LIN {X 0,Y 369.175,Z 240.992,A -85,B 0,C 180,E1 -12786.554,E2 -12786.554} C_VEL
LIN {X 0,Y 369.058,Z 241.013,A -85,B 0,C 180,E1 -12789.863,E2 -12789.863} C_VEL
LIN {X 0,Y 369.03,Z 241.015,A -85,B 0,C 180,E1 -12793.767,E2 -12793.767} C_VEL
LIN {X 0,Y 368.98,Z 241.021,A -85,B 0,C 180,E1 -12797.737,E2 -12797.737} C_VEL
LIN {X 0,Y 368.917,Z 241.027,A -85,B 0,C 180,E1 -12801.214,E2 -12801.214} C_VEL
LIN {X 0,Y 368.943,Z 241.021,A -85,B 0,C 180,E1 -12804.77,E2 -12804.77} C_VEL
LIN {X 0,Y 368.946,Z 241.015,A -85,B 0,C 180,E1 -12807.198,E2 -12807.198} C_VEL
LIN {X 0,Y 368.909,Z 241.02,A -85,B 0,C 180,E1 -12810.948,E2 -12810.948} C_VEL
LIN {X 0,Y 368.906,Z 241.024,A -85,B 0,C 180,E1 -12814.996,E2 -12814.996} C_VEL
LIN {X 0,Y 368.891,Z 241.027,A -85,B 0,C 180,E1 -12818.637,E2 -12818.637} C_VEL
LIN {X 0,Y 368.924,Z 241.033,A -85,B 0,C 180,E1 -12822.016,E2 -12822.016} C_VEL
LIN {X 0,Y 368.976,Z 241.248,A -85,B 0,C 180,E1 -12824.559,E2 -12824.559} C_VEL
LIN {X 0,Y 371.323,Z 251.732,A -85,B 0,C 180,E1 -12827.564,E2 -12827.564} C_VEL
LIN {X 0,Y 372.681,Z 259.06,A -85,B 0,C 180,E1 -12829.517,E2 -12829.517} C_VEL
LIN {X 0,Y 373.416,Z 261.979,A -85,B 0,C 180,E1 -12829.699,E2 -12829.699} C_VEL
LIN {X 0,Y 377.612,Z 280.099,A -85,B 0,C 180,E1 -12830.394,E2 -12830.394} C_VEL
LIN {X 0,Y 378.936,Z 287.781,A -85,B 0,C 180,E1 -12830.649,E2 -12830.649} C_VEL
LIN {X 0,Y 377.335,Z 366.53,A -85,B 0,C 180,E1 -12832.201,E2 -12832.201} C_VEL
LIN {X 0,Y 376.706,Z 379.905,A -85,B 0,C 180,E1 -12832.675,E2 -12832.675} C_VEL
LIN {X 0,Y 375.846,Z 392.955,A -85,B 0,C 180,E1 -12833.369,E2 -12833.369} C_VEL
LIN {X 0,Y 374.825,Z 404.268,A -85,B 0,C 180,E1 -12834.185,E2 -12834.185} C_VEL
LIN {X 0,Y 373.783,Z 414.895,A -85,B 0,C 180,E1 -12835.171,E2 -12835.171} C_VEL
LIN {X 0,Y 372.647,Z 424.936,A -85,B 0,C 180,E1 -12836.329,E2 -12836.329} C_VEL
LIN {X 0,Y 371.476,Z 434.527,A -85,B 0,C 180,E1 -12837.692,E2 -12837.692} C_VEL
LIN {X 0,Y 370.384,Z 443.005,A -85,B 0,C 180,E1 -12839.181,E2 -12839.181} C_VEL
LIN {X 0,Y 369.428,Z 450.372,A -85,B 0,C 180,E1 -12840.788,E2 -12840.788} C_VEL
LIN {X 0,Y 368.76,Z 455.563,A -85,B 0,C 180,E1 -12842.164,E2 -12842.164} C_VEL
LIN {X 0,Y 368.156,Z 460.932,A -85,B 0,C 180,E1 -12843.956,E2 -12843.956} C_VEL
LIN {X 0,Y 367.748,Z 464.988,A -85,B 0,C 180,E1 -12845.739,E2 -12845.739} C_VEL
LIN {X 0,Y 367.429,Z 467.852,A -85,B 0,C 180,E1 -12847.508,E2 -12847.508} C_VEL
LIN {X 0,Y 367.277,Z 469.892,A -85,B 0,C 180,E1 -12849.637,E2 -12849.637} C_VEL
LIN {X 0,Y 367.175,Z 470.375,A -85,B 0,C 180,E1 -12851.01,E2 -12851.01} C_VEL
LIN {X 0,Y 367.211,Z 469.971,A -85,B 0,C 180,E1 -12853.1,E2 -12853.1} C_VEL
LIN {X 0,Y 367.215,Z 468.91,A -85,B 0,C 180,E1 -12854.458,E2 -12854.458} C_VEL
LIN {X 0,Y 367.27,Z 467.556,A -85,B 0,C 180,E1 -12855.595,E2 -12855.595} C_VEL
LIN {X 0,Y 367.534,Z 464.884,A -85,B 0,C 180,E1 -12857.185,E2 -12857.185} C_VEL
LIN {X 0,Y 367.784,Z 460.721,A -85,B 0,C 180,E1 -12858.983,E2 -12858.983} C_VEL
LIN {X 0,Y 368.198,Z 454.637,A -85,B 0,C 180,E1 -12860.939,E2 -12860.939} C_VEL
LIN {X 0,Y 368.734,Z 448.069,A -85,B 0,C 180,E1 -12862.578,E2 -12862.578} C_VEL
LIN {X 0,Y 369.497,Z 439.608,A -85,B 0,C 180,E1 -12864.269,E2 -12864.269} C_VEL
LIN {X 0,Y 370.198,Z 431.102,A -85,B 0,C 180,E1 -12865.645,E2 -12865.645} C_VEL
LIN {X 0,Y 371.129,Z 420.552,A -85,B 0,C 180,E1 -12867.015,E2 -12867.015} C_VEL
LIN {X 0,Y 372.079,Z 409.847,A -85,B 0,C 180,E1 -12868.126,E2 -12868.126} C_VEL
LIN {X 0,Y 372.918,Z 398.589,A -85,B 0,C 180,E1 -12869.055,E2 -12869.055} C_VEL
LIN {X 0,Y 373.573,Z 386.78,A -85,B 0,C 180,E1 -12869.798,E2 -12869.798} C_VEL
LIN {X 0,Y 374.124,Z 374.049,A -85,B 0,C 180,E1 -12870.37,E2 -12870.37} C_VEL
LIN {X 0,Y 374.497,Z 360.971,A -85,B 0,C 180,E1 -12870.739,E2 -12870.739} C_VEL
LIN {X 0,Y 375.543,Z 284.816,A -85,B 0,C 180,E1 -12872.2,E2 -12872.2} C_VEL
LIN {X 0,Y 373.646,Z 274.125,A -85,B 0,C 180,E1 -12872.502,E2 -12872.502} C_VEL
LIN {X 0,Y 372.161,Z 268.743,A -85,B 0,C 180,E1 -12872.748,E2 -12872.748} C_VEL
LIN {X 0,Y 369.987,Z 263.95,A -85,B 0,C 180,E1 -12873.143,E2 -12873.143} C_VEL
LIN {X 0,Y 366.851,Z 258.406,A -85,B 0,C 180,E1 -12873.861,E2 -12873.861} C_VEL
LIN {X 0,Y 364.875,Z 254.78,A -85,B 0,C 180,E1 -12874.526,E2 -12874.526} C_VEL
LIN {X 0,Y 363.761,Z 251.58,A -85,B 0,C 180,E1 -12875.286,E2 -12875.286} C_VEL
LIN {X 0,Y 362.173,Z 242.319,A -85,B 0,C 180,E1 -12877.807,E2 -12877.807} C_VEL
LIN {X 0,Y 362.108,Z 241.901,A -85,B 0,C 180,E1 -12878.034,E2 -12878.034} C_VEL
LIN {X 0,Y 361.968,Z 241.897,A -85,B 0,C 180,E1 -12881.195,E2 -12881.195} C_VEL
LIN {X 0,Y 361.951,Z 241.896,A -85,B 0,C 180,E1 -12884.62,E2 -12884.62} C_VEL
LIN {X 0,Y 361.929,Z 241.891,A -85,B 0,C 180,E1 -12888.1,E2 -12888.1} C_VEL
LIN {X 0,Y 361.89,Z 241.904,A -85,B 0,C 180,E1 -12891.653,E2 -12891.653} C_VEL
LIN {X 0,Y 361.888,Z 241.886,A -85,B 0,C 180,E1 -12895.293,E2 -12895.293} C_VEL
LIN {X 0,Y 361.901,Z 241.889,A -85,B 0,C 180,E1 -12899.044,E2 -12899.044} C_VEL
LIN {X 0,Y 361.874,Z 241.912,A -85,B 0,C 180,E1 -12901.625,E2 -12901.625} C_VEL
LIN {X 0,Y 361.859,Z 241.901,A -85,B 0,C 180,E1 -12905.354,E2 -12905.354} C_VEL
LIN {X 0,Y 361.9,Z 241.903,A -85,B 0,C 180,E1 -12908.42,E2 -12908.42} C_VEL
LIN {X 0,Y 361.871,Z 241.9,A -85,B 0,C 180,E1 -12911.324,E2 -12911.324} C_VEL
LIN {X 0,Y 361.907,Z 241.9,A -85,B 0,C 180,E1 -12914.354,E2 -12914.354} C_VEL
LIN {X 0,Y 361.862,Z 241.909,A -85,B 0,C 180,E1 -12917.563,E2 -12917.563} C_VEL
LIN {X 0,Y 361.846,Z 241.888,A -85,B 0,C 180,E1 -12920.977,E2 -12920.977} C_VEL
LIN {X 0,Y 361.848,Z 241.91,A -85,B 0,C 180,E1 -12924.66,E2 -12924.66} C_VEL
LIN {X 0,Y 361.835,Z 241.91,A -85,B 0,C 180,E1 -12928.378,E2 -12928.378} C_VEL
LIN {X 0,Y 361.901,Z 241.877,A -85,B 0,C 180,E1 -12932.227,E2 -12932.227} C_VEL
LIN {X 0,Y 361.91,Z 241.89,A -85,B 0,C 180,E1 -12934.715,E2 -12934.715} C_VEL
LIN {X 0,Y 361.902,Z 241.908,A -85,B 0,C 180,E1 -12938.769,E2 -12938.769} C_VEL
LIN {X 0,Y 361.954,Z 241.884,A -85,B 0,C 180,E1 -12942.066,E2 -12942.066} C_VEL
LIN {X 0,Y 361.987,Z 241.868,A -85,B 0,C 180,E1 -12946.106,E2 -12946.106} C_VEL
LIN {X 0,Y 362.027,Z 241.885,A -85,B 0,C 180,E1 -12949.943,E2 -12949.943} C_VEL
LIN {X 0,Y 362.144,Z 241.87,A -85,B 0,C 180,E1 -12952.198,E2 -12952.198} C_VEL
LIN {X 0,Y 362.113,Z 241.867,A -85,B 0,C 180,E1 -12954.436,E2 -12954.436} C_VEL
LIN {X 0,Y 362.276,Z 241.826,A -85,B 0,C 180,E1 -12957.782,E2 -12957.782} C_VEL
LIN {X 0,Y 362.423,Z 241.823,A -85,B 0,C 180,E1 -12960.005,E2 -12960.005} C_VEL
LIN {X 0,Y 362.278,Z 241.855,A -85,B 0,C 180,E1 -12962.228,E2 -12962.228} C_VEL
LIN {X 0,Y 362.136,Z 241.866,A -85,B 0,C 180,E1 -12966.692,E2 -12966.692} C_VEL
LIN {X 0,Y 362.002,Z 241.865,A -85,B 0,C 180,E1 -12970.067,E2 -12970.067} C_VEL
LIN {X 0,Y 362.001,Z 241.886,A -85,B 0,C 180,E1 -12973.903,E2 -12973.903} C_VEL
LIN {X 0,Y 361.972,Z 241.893,A -85,B 0,C 180,E1 -12977.943,E2 -12977.943} C_VEL
LIN {X 0,Y 361.867,Z 241.889,A -85,B 0,C 180,E1 -12981.659,E2 -12981.659} C_VEL
LIN {X 0,Y 361.933,Z 241.9,A -85,B 0,C 180,E1 -12985.294,E2 -12985.294} C_VEL
LIN {X 0,Y 361.915,Z 241.897,A -85,B 0,C 180,E1 -12987.783,E2 -12987.783} C_VEL
LIN {X 0,Y 361.846,Z 241.908,A -85,B 0,C 180,E1 -12991.633,E2 -12991.633} C_VEL
LIN {X 0,Y 361.879,Z 241.905,A -85,B 0,C 180,E1 -12995.347,E2 -12995.347} C_VEL
LIN {X 0,Y 361.839,Z 241.91,A -85,B 0,C 180,E1 -12999.022,E2 -12999.022} C_VEL
LIN {X 0,Y 361.845,Z 241.901,A -85,B 0,C 180,E1 -13002.832,E2 -13002.832} C_VEL
LIN {X 0,Y 361.827,Z 241.886,A -85,B 0,C 180,E1 -13005.95,E2 -13005.95} C_VEL
LIN {X 0,Y 361.824,Z 241.914,A -85,B 0,C 180,E1 -13009.251,E2 -13009.251} C_VEL
LIN {X 0,Y 361.875,Z 241.903,A -85,B 0,C 180,E1 -13012.984,E2 -13012.984} C_VEL
LIN {X 0,Y 361.871,Z 241.908,A -85,B 0,C 180,E1 -13016.633,E2 -13016.633} C_VEL
LIN {X 0,Y 361.872,Z 241.911,A -85,B 0,C 180,E1 -13019.672,E2 -13019.672} C_VEL
LIN {X 0,Y 361.988,Z 242.11,A -85,B 0,C 180,E1 -13022.071,E2 -13022.071} C_VEL
LIN {X 0,Y 364.539,Z 255.351,A -85,B 0,C 180,E1 -13025.556,E2 -13025.556} C_VEL
LIN {X 0,Y 364.852,Z 258.893,A -85,B 0,C 180,E1 -13026.441,E2 -13026.441} C_VEL
LIN {X 0,Y 364.083,Z 268.447,A -85,B 0,C 180,E1 -13028.685,E2 -13028.685} C_VEL
LIN {X 0,Y 364.455,Z 271.791,A -85,B 0,C 180,E1 -13028.848,E2 -13028.848} C_VEL
LIN {X 0,Y 368.737,Z 299.58,A -85,B 0,C 180,E1 -13029.617,E2 -13029.617} C_VEL
LIN {X 0,Y 367.555,Z 376.344,A -85,B 0,C 180,E1 -13031.14,E2 -13031.14} C_VEL
LIN {X 0,Y 366.982,Z 389.637,A -85,B 0,C 180,E1 -13031.616,E2 -13031.616} C_VEL
LIN {X 0,Y 366.233,Z 401.838,A -85,B 0,C 180,E1 -13032.264,E2 -13032.264} C_VEL
LIN {X 0,Y 365.407,Z 413.34,A -85,B 0,C 180,E1 -13033.088,E2 -13033.088} C_VEL
LIN {X 0,Y 364.483,Z 425.147,A -85,B 0,C 180,E1 -13034.196,E2 -13034.196} C_VEL
LIN {X 0,Y 363.624,Z 435.74,A -85,B 0,C 180,E1 -13035.448,E2 -13035.448} C_VEL
LIN {X 0,Y 362.713,Z 445.257,A -85,B 0,C 180,E1 -13036.84,E2 -13036.84} C_VEL
LIN {X 0,Y 361.806,Z 454.405,A -85,B 0,C 180,E1 -13038.516,E2 -13038.516} C_VEL
LIN {X 0,Y 361.197,Z 461.769,A -85,B 0,C 180,E1 -13040.198,E2 -13040.198} C_VEL
LIN {X 0,Y 360.82,Z 466.746,A -85,B 0,C 180,E1 -13041.6,E2 -13041.6} C_VEL
LIN {X 0,Y 360.511,Z 471.567,A -85,B 0,C 180,E1 -13043.283,E2 -13043.283} C_VEL
LIN {X 0,Y 360.362,Z 475.253,A -85,B 0,C 180,E1 -13044.966,E2 -13044.966} C_VEL
LIN {X 0,Y 360.281,Z 477.91,A -85,B 0,C 180,E1 -13046.645,E2 -13046.645} C_VEL
LIN {X 0,Y 360.231,Z 479.16,A -85,B 0,C 180,E1 -13047.764,E2 -13047.764} C_VEL
LIN {X 0,Y 360.256,Z 480.002,A -85,B 0,C 180,E1 -13048.883,E2 -13048.883} C_VEL
LIN {X 0,Y 360.282,Z 480.408,A -85,B 0,C 180,E1 -13050,E2 -13050} C_VEL
LIN {X 0,Y 360.255,Z 480.427,A -85,B 0,C 180,E1 -13051.118,E2 -13051.118} C_VEL
LIN {X 0,Y 360.284,Z 479.31,A -85,B 0,C 180,E1 -13053.355,E2 -13053.355} C_VEL
LIN {X 0,Y 360.386,Z 478.118,A -85,B 0,C 180,E1 -13054.474,E2 -13054.474} C_VEL
LIN {X 0,Y 360.587,Z 474.517,A -85,B 0,C 180,E1 -13056.716,E2 -13056.716} C_VEL
LIN {X 0,Y 360.944,Z 470.633,A -85,B 0,C 180,E1 -13058.397,E2 -13058.397} C_VEL
LIN {X 0,Y 361.539,Z 465.636,A -85,B 0,C 180,E1 -13060.076,E2 -13060.076} C_VEL
LIN {X 0,Y 362.3,Z 459.377,A -85,B 0,C 180,E1 -13061.753,E2 -13061.753} C_VEL
LIN {X 0,Y 363.382,Z 451.556,A -85,B 0,C 180,E1 -13063.42,E2 -13063.42} C_VEL
LIN {X 0,Y 364.611,Z 442.258,A -85,B 0,C 180,E1 -13065.015,E2 -13065.015} C_VEL
LIN {X 0,Y 365.623,Z 433.19,A -85,B 0,C 180,E1 -13066.284,E2 -13066.284} C_VEL
LIN {X 0,Y 366.935,Z 423.186,A -85,B 0,C 180,E1 -13067.414,E2 -13067.414} C_VEL
LIN {X 0,Y 368.099,Z 412.726,A -85,B 0,C 180,E1 -13068.363,E2 -13068.363} C_VEL
LIN {X 0,Y 369.239,Z 400.178,A -85,B 0,C 180,E1 -13069.24,E2 -13069.24} C_VEL
LIN {X 0,Y 370.147,Z 387.693,A -85,B 0,C 180,E1 -13069.876,E2 -13069.876} C_VEL
LIN {X 0,Y 370.777,Z 374.729,A -85,B 0,C 180,E1 -13070.311,E2 -13070.311} C_VEL
LIN {X 0,Y 372.168,Z 299.835,A -85,B 0,C 180,E1 -13071.822,E2 -13071.822} C_VEL
LIN {X 0,Y 368.452,Z 280.07,A -85,B 0,C 180,E1 -13072.527,E2 -13072.527} C_VEL
LIN {X 0,Y 365.852,Z 268.462,A -85,B 0,C 180,E1 -13073.019,E2 -13073.019} C_VEL
LIN {X 0,Y 366.141,Z 265.039,A -85,B 0,C 180,E1 -13073.772,E2 -13073.772} C_VEL
LIN {X 0,Y 366.109,Z 261.48,A -85,B 0,C 180,E1 -13074.679,E2 -13074.679} C_VEL
LIN {X 0,Y 364.008,Z 250.919,A -85,B 0,C 180,E1 -13077.605,E2 -13077.605} C_VEL
LIN {X 0,Y 361.939,Z 242.037,A -85,B 0,C 180,E1 -13080.248,E2 -13080.248} C_VEL
LIN {X 0,Y 361.869,Z 241.911,A -85,B 0,C 180,E1 -13084.279,E2 -13084.279} C_VEL
LIN {X 0,Y 361.873,Z 241.909,A -85,B 0,C 180,E1 -13087.22,E2 -13087.22} C_VEL
LIN {X 0,Y 361.827,Z 241.915,A -85,B 0,C 180,E1 -13090.749,E2 -13090.749} C_VEL
LIN {X 0,Y 361.83,Z 241.913,A -85,B 0,C 180,E1 -13094.367,E2 -13094.367} C_VEL
LIN {X 0,Y 361.848,Z 241.893,A -85,B 0,C 180,E1 -13097.566,E2 -13097.566} C_VEL
LIN {X 0,Y 361.844,Z 241.908,A -85,B 0,C 180,E1 -13100.979,E2 -13100.979} C_VEL
LIN {X 0,Y 361.883,Z 241.904,A -85,B 0,C 180,E1 -13104.654,E2 -13104.654} C_VEL
LIN {X 0,Y 361.846,Z 241.905,A -85,B 0,C 180,E1 -13108.367,E2 -13108.367} C_VEL
LIN {X 0,Y 361.878,Z 241.905,A -85,B 0,C 180,E1 -13110.949,E2 -13110.949} C_VEL
LIN {X 0,Y 361.871,Z 241.909,A -85,B 0,C 180,E1 -13114.701,E2 -13114.701} C_VEL
LIN {X 0,Y 361.87,Z 241.906,A -85,B 0,C 180,E1 -13118.341,E2 -13118.341} C_VEL
LIN {X 0,Y 361.929,Z 241.9,A -85,B 0,C 180,E1 -13122.081,E2 -13122.081} C_VEL
LIN {X 0,Y 361.97,Z 241.889,A -85,B 0,C 180,E1 -13125.375,E2 -13125.375} C_VEL
LIN {X 0,Y 361.976,Z 241.887,A -85,B 0,C 180,E1 -13128.8,E2 -13128.8} C_VEL
LIN {X 0,Y 362.099,Z 241.878,A -85,B 0,C 180,E1 -13132.187,E2 -13132.187} C_VEL
LIN {X 0,Y 362.106,Z 241.874,A -85,B 0,C 180,E1 -13134.426,E2 -13134.426} C_VEL
LIN {X 0,Y 362.272,Z 241.854,A -85,B 0,C 180,E1 -13137.771,E2 -13137.771} C_VEL
LIN {X 0,Y 362.402,Z 241.841,A -85,B 0,C 180,E1 -13139.995,E2 -13139.995} C_VEL
LIN {X 0,Y 362.272,Z 241.853,A -85,B 0,C 180,E1 -13142.219,E2 -13142.219} C_VEL
LIN {X 0,Y 362.136,Z 241.868,A -85,B 0,C 180,E1 -13146.681,E2 -13146.681} C_VEL
LIN {X 0,Y 362.023,Z 241.891,A -85,B 0,C 180,E1 -13150.057,E2 -13150.057} C_VEL
LIN {X 0,Y 361.99,Z 241.893,A -85,B 0,C 180,E1 -13153.893,E2 -13153.893} C_VEL
LIN {X 0,Y 361.919,Z 241.904,A -85,B 0,C 180,E1 -13156.929,E2 -13156.929} C_VEL
LIN {X 0,Y 361.882,Z 241.908,A -85,B 0,C 180,E1 -13160.455,E2 -13160.455} C_VEL
LIN {X 0,Y 361.881,Z 241.906,A -85,B 0,C 180,E1 -13164.108,E2 -13164.108} C_VEL
LIN {X 0,Y 361.925,Z 241.884,A -85,B 0,C 180,E1 -13166.716,E2 -13166.716} C_VEL
LIN {X 0,Y 361.853,Z 241.902,A -85,B 0,C 180,E1 -13170.323,E2 -13170.323} C_VEL
LIN {X 0,Y 361.832,Z 241.909,A -85,B 0,C 180,E1 -13174.275,E2 -13174.275} C_VEL
LIN {X 0,Y 361.851,Z 241.91,A -85,B 0,C 180,E1 -13177.22,E2 -13177.22} C_VEL
LIN {X 0,Y 361.879,Z 241.903,A -85,B 0,C 180,E1 -13180.763,E2 -13180.763} C_VEL
LIN {X 0,Y 361.928,Z 242.099,A -85,B 0,C 180,E1 -13184.071,E2 -13184.071} C_VEL
LIN {X 0,Y 364.016,Z 251.258,A -85,B 0,C 180,E1 -13186.778,E2 -13186.778} C_VEL
LIN {X 0,Y 365.668,Z 259.324,A -85,B 0,C 180,E1 -13188.99,E2 -13188.99} C_VEL
LIN {X 0,Y 367.337,Z 264.457,A -85,B 0,C 180,E1 -13189.28,E2 -13189.28} C_VEL
LIN {X 0,Y 371.361,Z 281.98,A -85,B 0,C 180,E1 -13189.972,E2 -13189.972} C_VEL
LIN {X 0,Y 372.513,Z 288.031,A -85,B 0,C 180,E1 -13190.188,E2 -13190.188} C_VEL
LIN {X 0,Y 370.835,Z 366.571,A -85,B 0,C 180,E1 -13191.764,E2 -13191.764} C_VEL
LIN {X 0,Y 370.177,Z 379.944,A -85,B 0,C 180,E1 -13192.245,E2 -13192.245} C_VEL
LIN {X 0,Y 369.34,Z 391.948,A -85,B 0,C 180,E1 -13192.885,E2 -13192.885} C_VEL
LIN {X 0,Y 368.287,Z 403.751,A -85,B 0,C 180,E1 -13193.731,E2 -13193.731} C_VEL
LIN {X 0,Y 367.13,Z 414.957,A -85,B 0,C 180,E1 -13194.782,E2 -13194.782} C_VEL
LIN {X 0,Y 365.735,Z 426.361,A -85,B 0,C 180,E1 -13196.133,E2 -13196.133} C_VEL
LIN {X 0,Y 364.508,Z 435.985,A -85,B 0,C 180,E1 -13197.572,E2 -13197.572} C_VEL
LIN {X 0,Y 363.319,Z 444.544,A -85,B 0,C 180,E1 -13199.162,E2 -13199.162} C_VEL
LIN {X 0,Y 362.23,Z 452.394,A -85,B 0,C 180,E1 -13200.984,E2 -13200.984} C_VEL
LIN {X 0,Y 361.433,Z 458.505,A -85,B 0,C 180,E1 -13202.809,E2 -13202.809} C_VEL
LIN {X 0,Y 360.909,Z 463.203,A -85,B 0,C 180,E1 -13204.633,E2 -13204.633} C_VEL
LIN {X 0,Y 360.543,Z 466.505,A -85,B 0,C 180,E1 -13206.353,E2 -13206.353} C_VEL
LIN {X 0,Y 360.233,Z 468.962,A -85,B 0,C 180,E1 -13208.242,E2 -13208.242} C_VEL
LIN {X 0,Y 360.189,Z 469.949,A -85,B 0,C 180,E1 -13209.463,E2 -13209.463} C_VEL
LIN {X 0,Y 360.092,Z 470.433,A -85,B 0,C 180,E1 -13210.622,E2 -13210.622} C_VEL
LIN {X 0,Y 360.058,Z 470.477,A -85,B 0,C 180,E1 -13211.801,E2 -13211.801} C_VEL
LIN {X 0,Y 360.101,Z 470.105,A -85,B 0,C 180,E1 -13212.977,E2 -13212.977} C_VEL
LIN {X 0,Y 360.121,Z 469.309,A -85,B 0,C 180,E1 -13214.144,E2 -13214.144} C_VEL
LIN {X 0,Y 360.169,Z 468.041,A -85,B 0,C 180,E1 -13215.305,E2 -13215.305} C_VEL
LIN {X 0,Y 360.43,Z 465.192,A -85,B 0,C 180,E1 -13217.113,E2 -13217.113} C_VEL
LIN {X 0,Y 360.659,Z 461.569,A -85,B 0,C 180,E1 -13218.763,E2 -13218.763} C_VEL
LIN {X 0,Y 360.96,Z 456.663,A -85,B 0,C 180,E1 -13220.474,E2 -13220.474} C_VEL
LIN {X 0,Y 361.609,Z 449.814,A -85,B 0,C 180,E1 -13222.337,E2 -13222.337} C_VEL
LIN {X 0,Y 362.215,Z 442.733,A -85,B 0,C 180,E1 -13223.874,E2 -13223.874} C_VEL
LIN {X 0,Y 362.877,Z 434.836,A -85,B 0,C 180,E1 -13225.278,E2 -13225.278} C_VEL
LIN {X 0,Y 363.787,Z 425.158,A -85,B 0,C 180,E1 -13226.677,E2 -13226.677} C_VEL
LIN {X 0,Y 364.814,Z 414.258,A -85,B 0,C 180,E1 -13227.943,E2 -13227.943} C_VEL
LIN {X 0,Y 365.749,Z 402.902,A -85,B 0,C 180,E1 -13228.986,E2 -13228.986} C_VEL
LIN {X 0,Y 366.505,Z 390.434,A -85,B 0,C 180,E1 -13229.862,E2 -13229.862} C_VEL
LIN {X 0,Y 367.136,Z 377.712,A -85,B 0,C 180,E1 -13230.514,E2 -13230.514} C_VEL
LIN {X 0,Y 367.593,Z 365.51,A -85,B 0,C 180,E1 -13230.924,E2 -13230.924} C_VEL
LIN {X 0,Y 368.867,Z 286.373,A -85,B 0,C 180,E1 -13232.484,E2 -13232.484} C_VEL
LIN {X 0,Y 364.244,Z 259.612,A -85,B 0,C 180,E1 -13233.287,E2 -13233.287} C_VEL
LIN {X 0,Y 364.446,Z 256.919,A -85,B 0,C 180,E1 -13233.87,E2 -13233.87} C_VEL
LIN {X 0,Y 363.964,Z 252.7,A -85,B 0,C 180,E1 -13234.985,E2 -13234.985} C_VEL
LIN {X 0,Y 363.761,Z 251.58,A -85,B 0,C 180,E1 -13235.286,E2 -13235.286} C_VEL
LIN {X 0,Y 362.739,Z 249.786,A -85,B 0,C 180,E1 -13235.816,E2 -13235.816} C_VEL
LIN {X 0,Y 356.039,Z 244.929,A -85,B 0,C 180,E1 -13237.513,E2 -13237.513} C_VEL
LIN {X 0,Y 355.136,Z 243.116,A -85,B 0,C 180,E1 -13238.082,E2 -13238.082} C_VEL
LIN {X 0,Y 355.06,Z 242.774,A -85,B 0,C 180,E1 -13238.288,E2 -13238.288} C_VEL
LIN {X 0,Y 354.927,Z 242.773,A -85,B 0,C 180,E1 -13241.42,E2 -13241.42} C_VEL
LIN {X 0,Y 354.899,Z 242.774,A -85,B 0,C 180,E1 -13244.918,E2 -13244.918} C_VEL
LIN {X 0,Y 354.872,Z 242.765,A -85,B 0,C 180,E1 -13248.473,E2 -13248.473} C_VEL
LIN {X 0,Y 354.858,Z 242.78,A -85,B 0,C 180,E1 -13252.104,E2 -13252.104} C_VEL
LIN {X 0,Y 354.858,Z 242.757,A -85,B 0,C 180,E1 -13255.83,E2 -13255.83} C_VEL
LIN {X 0,Y 354.824,Z 242.78,A -85,B 0,C 180,E1 -13259.681,E2 -13259.681} C_VEL
LIN {X 0,Y 354.801,Z 242.789,A -85,B 0,C 180,E1 -13262.331,E2 -13262.331} C_VEL
LIN {X 0,Y 354.81,Z 242.78,A -85,B 0,C 180,E1 -13265.709,E2 -13265.709} C_VEL
LIN {X 0,Y 354.864,Z 242.782,A -85,B 0,C 180,E1 -13269.327,E2 -13269.327} C_VEL
LIN {X 0,Y 354.81,Z 242.77,A -85,B 0,C 180,E1 -13272.881,E2 -13272.881} C_VEL
LIN {X 0,Y 354.841,Z 242.786,A -85,B 0,C 180,E1 -13276.125,E2 -13276.125} C_VEL
LIN {X 0,Y 354.827,Z 242.777,A -85,B 0,C 180,E1 -13279.194,E2 -13279.194} C_VEL
LIN {X 0,Y 354.785,Z 242.773,A -85,B 0,C 180,E1 -13282.406,E2 -13282.406} C_VEL
LIN {X 0,Y 354.786,Z 242.787,A -85,B 0,C 180,E1 -13284.946,E2 -13284.946} C_VEL
LIN {X 0,Y 354.791,Z 242.787,A -85,B 0,C 180,E1 -13288.405,E2 -13288.405} C_VEL
LIN {X 0,Y 354.832,Z 242.759,A -85,B 0,C 180,E1 -13291.625,E2 -13291.625} C_VEL
LIN {X 0,Y 354.88,Z 242.759,A -85,B 0,C 180,E1 -13294.178,E2 -13294.178} C_VEL
LIN {X 0,Y 354.833,Z 242.782,A -85,B 0,C 180,E1 -13297.9,E2 -13297.9} C_VEL
LIN {X 0,Y 354.909,Z 242.761,A -85,B 0,C 180,E1 -13301.896,E2 -13301.896} C_VEL
LIN {X 0,Y 354.932,Z 242.747,A -85,B 0,C 180,E1 -13305.986,E2 -13305.986} C_VEL
LIN {X 0,Y 354.974,Z 242.765,A -85,B 0,C 180,E1 -13309.741,E2 -13309.741} C_VEL
LIN {X 0,Y 355.106,Z 242.747,A -85,B 0,C 180,E1 -13312.042,E2 -13312.042} C_VEL
LIN {X 0,Y 355.087,Z 242.742,A -85,B 0,C 180,E1 -13314.326,E2 -13314.326} C_VEL
LIN {X 0,Y 355.239,Z 242.702,A -85,B 0,C 180,E1 -13317.738,E2 -13317.738} C_VEL
LIN {X 0,Y 355.371,Z 242.701,A -85,B 0,C 180,E1 -13320.005,E2 -13320.005} C_VEL
LIN {X 0,Y 355.241,Z 242.731,A -85,B 0,C 180,E1 -13322.273,E2 -13322.273} C_VEL
LIN {X 0,Y 355.1,Z 242.742,A -85,B 0,C 180,E1 -13326.825,E2 -13326.825} C_VEL
LIN {X 0,Y 354.958,Z 242.742,A -85,B 0,C 180,E1 -13330.269,E2 -13330.269} C_VEL
LIN {X 0,Y 354.946,Z 242.766,A -85,B 0,C 180,E1 -13334.023,E2 -13334.023} C_VEL
LIN {X 0,Y 354.928,Z 242.77,A -85,B 0,C 180,E1 -13338.113,E2 -13338.113} C_VEL
LIN {X 0,Y 354.821,Z 242.768,A -85,B 0,C 180,E1 -13342.111,E2 -13342.111} C_VEL
LIN {X 0,Y 354.905,Z 242.775,A -85,B 0,C 180,E1 -13345.831,E2 -13345.831} C_VEL
LIN {X 0,Y 354.813,Z 242.769,A -85,B 0,C 180,E1 -13349.687,E2 -13349.687} C_VEL
LIN {X 0,Y 354.824,Z 242.787,A -85,B 0,C 180,E1 -13353.687,E2 -13353.687} C_VEL
LIN {X 0,Y 354.802,Z 242.783,A -85,B 0,C 180,E1 -13356.463,E2 -13356.463} C_VEL
LIN {X 0,Y 354.809,Z 242.791,A -85,B 0,C 180,E1 -13359.422,E2 -13359.422} C_VEL
LIN {X 0,Y 354.797,Z 242.778,A -85,B 0,C 180,E1 -13362.87,E2 -13362.87} C_VEL
LIN {X 0,Y 354.776,Z 242.766,A -85,B 0,C 180,E1 -13366.106,E2 -13366.106} C_VEL
LIN {X 0,Y 354.777,Z 242.791,A -85,B 0,C 180,E1 -13369.178,E2 -13369.178} C_VEL
LIN {X 0,Y 354.812,Z 242.78,A -85,B 0,C 180,E1 -13372.407,E2 -13372.407} C_VEL
LIN {X 0,Y 354.824,Z 242.784,A -85,B 0,C 180,E1 -13374.943,E2 -13374.943} C_VEL
LIN {X 0,Y 354.805,Z 242.786,A -85,B 0,C 180,E1 -13378.407,E2 -13378.407} C_VEL
LIN {X 0,Y 354.927,Z 242.945,A -85,B 0,C 180,E1 -13381.8,E2 -13381.8} C_VEL
LIN {X 0,Y 356.95,Z 253.585,A -85,B 0,C 180,E1 -13384.676,E2 -13384.676} C_VEL
LIN {X 0,Y 357.87,Z 259.691,A -85,B 0,C 180,E1 -13386.261,E2 -13386.261} C_VEL
LIN {X 0,Y 357.185,Z 268.454,A -85,B 0,C 180,E1 -13388.351,E2 -13388.351} C_VEL
LIN {X 0,Y 357.698,Z 272.545,A -85,B 0,C 180,E1 -13388.526,E2 -13388.526} C_VEL
LIN {X 0,Y 361.962,Z 301.104,A -85,B 0,C 180,E1 -13389.329,E2 -13389.329} C_VEL
LIN {X 0,Y 360.728,Z 376.236,A -85,B 0,C 180,E1 -13390.843,E2 -13390.843} C_VEL
LIN {X 0,Y 360.138,Z 389.531,A -85,B 0,C 180,E1 -13391.328,E2 -13391.328} C_VEL
LIN {X 0,Y 359.371,Z 401.734,A -85,B 0,C 180,E1 -13391.987,E2 -13391.987} C_VEL
LIN {X 0,Y 358.438,Z 414.047,A -85,B 0,C 180,E1 -13392.896,E2 -13392.896} C_VEL
LIN {X 0,Y 357.495,Z 425.696,A -85,B 0,C 180,E1 -13394.025,E2 -13394.025} C_VEL
LIN {X 0,Y 356.607,Z 436.178,A -85,B 0,C 180,E1 -13395.302,E2 -13395.302} C_VEL
LIN {X 0,Y 355.748,Z 444.724,A -85,B 0,C 180,E1 -13396.578,E2 -13396.578} C_VEL
LIN {X 0,Y 354.787,Z 453.962,A -85,B 0,C 180,E1 -13398.285,E2 -13398.285} C_VEL
LIN {X 0,Y 354.157,Z 461.388,A -85,B 0,C 180,E1 -13400.001,E2 -13400.001} C_VEL
LIN {X 0,Y 353.756,Z 466.418,A -85,B 0,C 180,E1 -13401.431,E2 -13401.431} C_VEL
LIN {X 0,Y 353.43,Z 471.289,A -85,B 0,C 180,E1 -13403.148,E2 -13403.148} C_VEL
LIN {X 0,Y 353.266,Z 475.021,A -85,B 0,C 180,E1 -13404.864,E2 -13404.864} C_VEL
LIN {X 0,Y 353.205,Z 477.722,A -85,B 0,C 180,E1 -13406.578,E2 -13406.578} C_VEL
LIN {X 0,Y 353.156,Z 479.864,A -85,B 0,C 180,E1 -13408.86,E2 -13408.86} C_VEL
LIN {X 0,Y 353.183,Z 480.299,A -85,B 0,C 180,E1 -13410,E2 -13410} C_VEL
LIN {X 0,Y 353.155,Z 480.338,A -85,B 0,C 180,E1 -13411.141,E2 -13411.141} C_VEL
LIN {X 0,Y 353.21,Z 479.266,A -85,B 0,C 180,E1 -13413.423,E2 -13413.423} C_VEL
LIN {X 0,Y 353.302,Z 478.108,A -85,B 0,C 180,E1 -13414.564,E2 -13414.564} C_VEL
LIN {X 0,Y 353.521,Z 474.549,A -85,B 0,C 180,E1 -13416.851,E2 -13416.851} C_VEL
LIN {X 0,Y 353.921,Z 470.708,A -85,B 0,C 180,E1 -13418.565,E2 -13418.565} C_VEL
LIN {X 0,Y 354.55,Z 465.758,A -85,B 0,C 180,E1 -13420.277,E2 -13420.277} C_VEL
LIN {X 0,Y 355.346,Z 459.552,A -85,B 0,C 180,E1 -13421.986,E2 -13421.986} C_VEL
LIN {X 0,Y 356.487,Z 451.818,A -85,B 0,C 180,E1 -13423.685,E2 -13423.685} C_VEL
LIN {X 0,Y 357.747,Z 442.831,A -85,B 0,C 180,E1 -13425.271,E2 -13425.271} C_VEL
LIN {X 0,Y 358.842,Z 433.631,A -85,B 0,C 180,E1 -13426.601,E2 -13426.601} C_VEL
LIN {X 0,Y 360.202,Z 423.754,A -85,B 0,C 180,E1 -13427.75,E2 -13427.75} C_VEL
LIN {X 0,Y 361.409,Z 413.501,A -85,B 0,C 180,E1 -13428.715,E2 -13428.715} C_VEL
LIN {X 0,Y 362.607,Z 401.273,A -85,B 0,C 180,E1 -13429.606,E2 -13429.606} C_VEL
LIN {X 0,Y 363.576,Z 388.474,A -85,B 0,C 180,E1 -13430.288,E2 -13430.288} C_VEL
LIN {X 0,Y 364.257,Z 376.163,A -85,B 0,C 180,E1 -13430.728,E2 -13430.728} C_VEL
LIN {X 0,Y 365.781,Z 300.95,A -85,B 0,C 180,E1 -13432.278,E2 -13432.278} C_VEL
LIN {X 0,Y 362.169,Z 281.629,A -85,B 0,C 180,E1 -13432.987,E2 -13432.987} C_VEL
LIN {X 0,Y 359.149,Z 268.362,A -85,B 0,C 180,E1 -13433.565,E2 -13433.565} C_VEL
LIN {X 0,Y 359.368,Z 264.123,A -85,B 0,C 180,E1 -13434.556,E2 -13434.556} C_VEL
LIN {X 0,Y 357.652,Z 254.814,A -85,B 0,C 180,E1 -13437.162,E2 -13437.162} C_VEL
LIN {X 0,Y 355.202,Z 244.239,A -85,B 0,C 180,E1 -13440.3,E2 -13440.3} C_VEL
LIN {X 0,Y 354.84,Z 242.816,A -85,B 0,C 180,E1 -13440.83,E2 -13440.83} C_VEL
LIN {X 0,Y 354.822,Z 242.784,A -85,B 0,C 180,E1 -13443.701,E2 -13443.701} C_VEL
LIN {X 0,Y 354.81,Z 242.786,A -85,B 0,C 180,E1 -13446.458,E2 -13446.458} C_VEL
LIN {X 0,Y 354.783,Z 242.784,A -85,B 0,C 180,E1 -13449.411,E2 -13449.411} C_VEL
LIN {X 0,Y 354.799,Z 242.777,A -85,B 0,C 180,E1 -13452.864,E2 -13452.864} C_VEL
LIN {X 0,Y 354.78,Z 242.784,A -85,B 0,C 180,E1 -13456.101,E2 -13456.101} C_VEL
LIN {X 0,Y 354.799,Z 242.789,A -85,B 0,C 180,E1 -13459.176,E2 -13459.176} C_VEL
LIN {X 0,Y 354.813,Z 242.786,A -85,B 0,C 180,E1 -13462.402,E2 -13462.402} C_VEL
LIN {X 0,Y 354.82,Z 242.784,A -85,B 0,C 180,E1 -13464.937,E2 -13464.937} C_VEL
LIN {X 0,Y 354.802,Z 242.782,A -85,B 0,C 180,E1 -13468.403,E2 -13468.403} C_VEL
LIN {X 0,Y 354.808,Z 242.781,A -85,B 0,C 180,E1 -13471.611,E2 -13471.611} C_VEL
LIN {X 0,Y 354.814,Z 242.781,A -85,B 0,C 180,E1 -13475.416,E2 -13475.416} C_VEL
LIN {X 0,Y 354.835,Z 242.782,A -85,B 0,C 180,E1 -13479.109,E2 -13479.109} C_VEL
LIN {X 0,Y 354.889,Z 242.777,A -85,B 0,C 180,E1 -13482.715,E2 -13482.715} C_VEL
LIN {X 0,Y 354.959,Z 242.768,A -85,B 0,C 180,E1 -13486.251,E2 -13486.251} C_VEL
LIN {X 0,Y 354.961,Z 242.762,A -85,B 0,C 180,E1 -13489.731,E2 -13489.731} C_VEL
LIN {X 0,Y 355.11,Z 242.746,A -85,B 0,C 180,E1 -13493.175,E2 -13493.175} C_VEL
LIN {X 0,Y 355.234,Z 242.73,A -85,B 0,C 180,E1 -13497.727,E2 -13497.727} C_VEL
LIN {X 0,Y 355.353,Z 242.719,A -85,B 0,C 180,E1 -13499.995,E2 -13499.995} C_VEL
LIN {X 0,Y 355.234,Z 242.728,A -85,B 0,C 180,E1 -13502.262,E2 -13502.262} C_VEL
LIN {X 0,Y 355.1,Z 242.743,A -85,B 0,C 180,E1 -13506.814,E2 -13506.814} C_VEL
LIN {X 0,Y 354.97,Z 242.768,A -85,B 0,C 180,E1 -13510.259,E2 -13510.259} C_VEL
LIN {X 0,Y 354.935,Z 242.773,A -85,B 0,C 180,E1 -13514.013,E2 -13514.013} C_VEL
LIN {X 0,Y 354.879,Z 242.778,A -85,B 0,C 180,E1 -13518.086,E2 -13518.086} C_VEL
LIN {X 0,Y 354.822,Z 242.781,A -85,B 0,C 180,E1 -13522.1,E2 -13522.1} C_VEL
LIN {X 0,Y 354.883,Z 242.761,A -85,B 0,C 180,E1 -13525.822,E2 -13525.822} C_VEL
LIN {X 0,Y 354.799,Z 242.785,A -85,B 0,C 180,E1 -13529.676,E2 -13529.676} C_VEL
LIN {X 0,Y 354.784,Z 242.79,A -85,B 0,C 180,E1 -13533.696,E2 -13533.696} C_VEL
LIN {X 0,Y 354.78,Z 242.792,A -85,B 0,C 180,E1 -13536.453,E2 -13536.453} C_VEL
LIN {X 0,Y 354.799,Z 242.79,A -85,B 0,C 180,E1 -13539.418,E2 -13539.418} C_VEL
LIN {X 0,Y 354.83,Z 242.783,A -85,B 0,C 180,E1 -13542.874,E2 -13542.874} C_VEL
LIN {X 0,Y 354.903,Z 243.018,A -85,B 0,C 180,E1 -13543.589,E2 -13543.589} C_VEL
LIN {X 0,Y 357.062,Z 252.501,A -85,B 0,C 180,E1 -13546.457,E2 -13546.457} C_VEL
LIN {X 0,Y 358.533,Z 259.431,A -85,B 0,C 180,E1 -13548.402,E2 -13548.402} C_VEL
LIN {X 0,Y 360.839,Z 265.481,A -85,B 0,C 180,E1 -13548.779,E2 -13548.779} C_VEL
LIN {X 0,Y 364.861,Z 282.541,A -85,B 0,C 180,E1 -13549.484,E2 -13549.484} C_VEL
LIN {X 0,Y 366.103,Z 289.065,A -85,B 0,C 180,E1 -13549.724,E2 -13549.724} C_VEL
LIN {X 0,Y 364.373,Z 366.84,A -85,B 0,C 180,E1 -13551.314,E2 -13551.314} C_VEL
LIN {X 0,Y 363.691,Z 380.152,A -85,B 0,C 180,E1 -13551.802,E2 -13551.802} C_VEL
LIN {X 0,Y 362.731,Z 393.202,A -85,B 0,C 180,E1 -13552.519,E2 -13552.519} C_VEL
LIN {X 0,Y 361.488,Z 405.594,A -85,B 0,C 180,E1 -13553.458,E2 -13553.458} C_VEL
LIN {X 0,Y 360.206,Z 417.289,A -85,B 0,C 180,E1 -13554.619,E2 -13554.619} C_VEL
LIN {X 0,Y 358.862,Z 427.57,A -85,B 0,C 180,E1 -13555.903,E2 -13555.903} C_VEL
LIN {X 0,Y 357.664,Z 436.404,A -85,B 0,C 180,E1 -13557.273,E2 -13557.273} C_VEL
LIN {X 0,Y 356.467,Z 444.617,A -85,B 0,C 180,E1 -13558.833,E2 -13558.833} C_VEL
LIN {X 0,Y 355.302,Z 452.643,A -85,B 0,C 180,E1 -13560.735,E2 -13560.735} C_VEL
LIN {X 0,Y 354.592,Z 457.679,A -85,B 0,C 180,E1 -13562.24,E2 -13562.24} C_VEL
LIN {X 0,Y 353.977,Z 462.623,A -85,B 0,C 180,E1 -13564.1,E2 -13564.1} C_VEL
LIN {X 0,Y 353.49,Z 466.538,A -85,B 0,C 180,E1 -13566.124,E2 -13566.124} C_VEL
LIN {X 0,Y 353.207,Z 468.761,A -85,B 0,C 180,E1 -13567.786,E2 -13567.786} C_VEL
LIN {X 0,Y 353.11,Z 470.006,A -85,B 0,C 180,E1 -13569.279,E2 -13569.279} C_VEL
LIN {X 0,Y 352.956,Z 470.621,A -85,B 0,C 180,E1 -13571.422,E2 -13571.422} C_VEL
LIN {X 0,Y 353.01,Z 470.24,A -85,B 0,C 180,E1 -13572.84,E2 -13572.84} C_VEL
LIN {X 0,Y 353.044,Z 468.519,A -85,B 0,C 180,E1 -13575.001,E2 -13575.001} C_VEL
LIN {X 0,Y 353.332,Z 465.494,A -85,B 0,C 180,E1 -13577.035,E2 -13577.035} C_VEL
LIN {X 0,Y 353.613,Z 460.942,A -85,B 0,C 180,E1 -13579.116,E2 -13579.116} C_VEL
LIN {X 0,Y 353.995,Z 455.837,A -85,B 0,C 180,E1 -13580.861,E2 -13580.861} C_VEL
LIN {X 0,Y 354.592,Z 449.515,A -85,B 0,C 180,E1 -13582.57,E2 -13582.57} C_VEL
LIN {X 0,Y 355.323,Z 441.343,A -85,B 0,C 180,E1 -13584.324,E2 -13584.324} C_VEL
LIN {X 0,Y 356.032,Z 433.143,A -85,B 0,C 180,E1 -13585.754,E2 -13585.754} C_VEL
LIN {X 0,Y 357.017,Z 423.105,A -85,B 0,C 180,E1 -13587.179,E2 -13587.179} C_VEL
LIN {X 0,Y 358.054,Z 412.586,A -85,B 0,C 180,E1 -13588.369,E2 -13588.369} C_VEL
LIN {X 0,Y 358.94,Z 401.659,A -85,B 0,C 180,E1 -13589.354,E2 -13589.354} C_VEL
LIN {X 0,Y 359.727,Z 389.395,A -85,B 0,C 180,E1 -13590.21,E2 -13590.21} C_VEL
LIN {X 0,Y 360.28,Z 377.835,A -85,B 0,C 180,E1 -13590.803,E2 -13590.803} C_VEL
LIN {X 0,Y 360.743,Z 364.45,A -85,B 0,C 180,E1 -13591.25,E2 -13591.25} C_VEL
LIN {X 0,Y 362.08,Z 287.214,A -85,B 0,C 180,E1 -13592.799,E2 -13592.799} C_VEL
LIN {X 0,Y 357.38,Z 259.78,A -85,B 0,C 180,E1 -13593.629,E2 -13593.629} C_VEL
LIN {X 0,Y 357.452,Z 258.137,A -85,B 0,C 180,E1 -13593.946,E2 -13593.946} C_VEL
LIN {X 0,Y 356.976,Z 253.888,A -85,B 0,C 180,E1 -13595.082,E2 -13595.082} C_VEL
LIN {X 0,Y 355.395,Z 244.502,A -85,B 0,C 180,E1 -13597.67,E2 -13597.67} C_VEL
LIN {X 0,Y 355.136,Z 243.116,A -85,B 0,C 180,E1 -13598.082,E2 -13598.082} C_VEL
LIN {X 0,Y 354.808,Z 242.788,A -85,B 0,C 180,E1 -13598.52,E2 -13598.52} C_VEL
LIN {X 0,Y 352.554,Z 243.069,A -85,B 0,C 180,E1 -13599.89,E2 -13599.89} C_VEL
LIN {X 0,Y 348.94,Z 243.698,A -85,B 0,C 180,E1 -13601.774,E2 -13601.774} C_VEL
LIN {X 0,Y 347.953,Z 243.662,A -85,B 0,C 180,E1 -13602.761,E2 -13602.761} C_VEL
LIN {X 0,Y 347.877,Z 243.651,A -85,B 0,C 180,E1 -13603.095,E2 -13603.095} C_VEL
LIN {X 0,Y 347.815,Z 243.661,A -85,B 0,C 180,E1 -13606.432,E2 -13606.432} C_VEL
LIN {X 0,Y 347.822,Z 243.639,A -85,B 0,C 180,E1 -13608.862,E2 -13608.862} C_VEL
LIN {X 0,Y 347.808,Z 243.66,A -85,B 0,C 180,E1 -13612.576,E2 -13612.576} C_VEL
LIN {X 0,Y 347.79,Z 243.631,A -85,B 0,C 180,E1 -13616.395,E2 -13616.395} C_VEL
LIN {X 0,Y 347.757,Z 243.662,A -85,B 0,C 180,E1 -13620.347,E2 -13620.347} C_VEL
LIN {X 0,Y 347.746,Z 243.671,A -85,B 0,C 180,E1 -13623.07,E2 -13623.07} C_VEL
LIN {X 0,Y 347.771,Z 243.659,A -85,B 0,C 180,E1 -13626.078,E2 -13626.078} C_VEL
LIN {X 0,Y 347.789,Z 243.66,A -85,B 0,C 180,E1 -13628.787,E2 -13628.787} C_VEL
LIN {X 0,Y 347.788,Z 243.647,A -85,B 0,C 180,E1 -13631.824,E2 -13631.824} C_VEL
LIN {X 0,Y 347.818,Z 243.653,A -85,B 0,C 180,E1 -13635.007,E2 -13635.007} C_VEL
LIN {X 0,Y 347.756,Z 243.66,A -85,B 0,C 180,E1 -13638.395,E2 -13638.395} C_VEL
LIN {X 0,Y 347.751,Z 243.644,A -85,B 0,C 180,E1 -13642.015,E2 -13642.015} C_VEL
LIN {X 0,Y 347.718,Z 243.667,A -85,B 0,C 180,E1 -13645.541,E2 -13645.541} C_VEL
LIN {X 0,Y 347.74,Z 243.667,A -85,B 0,C 180,E1 -13648.308,E2 -13648.308} C_VEL
LIN {X 0,Y 347.784,Z 243.638,A -85,B 0,C 180,E1 -13650.996,E2 -13650.996} C_VEL
LIN {X 0,Y 347.812,Z 243.637,A -85,B 0,C 180,E1 -13653.613,E2 -13653.613} C_VEL
LIN {X 0,Y 347.779,Z 243.656,A -85,B 0,C 180,E1 -13656.168,E2 -13656.168} C_VEL
LIN {X 0,Y 347.82,Z 243.654,A -85,B 0,C 180,E1 -13659.916,E2 -13659.916} C_VEL
LIN {X 0,Y 347.853,Z 243.641,A -85,B 0,C 180,E1 -13662.365,E2 -13662.365} C_VEL
LIN {X 0,Y 347.886,Z 243.624,A -85,B 0,C 180,E1 -13665.976,E2 -13665.976} C_VEL
LIN {X 0,Y 347.924,Z 243.645,A -85,B 0,C 180,E1 -13669.531,E2 -13669.531} C_VEL
LIN {X 0,Y 348.067,Z 243.625,A -85,B 0,C 180,E1 -13671.88,E2 -13671.88} C_VEL
LIN {X 0,Y 348.062,Z 243.617,A -85,B 0,C 180,E1 -13674.211,E2 -13674.211} C_VEL
LIN {X 0,Y 348.201,Z 243.577,A -85,B 0,C 180,E1 -13677.692,E2 -13677.692} C_VEL
LIN {X 0,Y 348.322,Z 243.578,A -85,B 0,C 180,E1 -13680.005,E2 -13680.005} C_VEL
LIN {X 0,Y 348.204,Z 243.608,A -85,B 0,C 180,E1 -13682.319,E2 -13682.319} C_VEL
LIN {X 0,Y 348.068,Z 243.618,A -85,B 0,C 180,E1 -13686.963,E2 -13686.963} C_VEL
LIN {X 0,Y 347.898,Z 243.621,A -85,B 0,C 180,E1 -13690.48,E2 -13690.48} C_VEL
LIN {X 0,Y 347.902,Z 243.644,A -85,B 0,C 180,E1 -13694.154,E2 -13694.154} C_VEL
LIN {X 0,Y 347.896,Z 243.643,A -85,B 0,C 180,E1 -13698.294,E2 -13698.294} C_VEL
LIN {X 0,Y 347.773,Z 243.643,A -85,B 0,C 180,E1 -13701.63,E2 -13701.63} C_VEL
LIN {X 0,Y 347.818,Z 243.66,A -85,B 0,C 180,E1 -13705.112,E2 -13705.112} C_VEL
LIN {X 0,Y 347.809,Z 243.654,A -85,B 0,C 180,E1 -13707.698,E2 -13707.698} C_VEL
LIN {X 0,Y 347.753,Z 243.663,A -85,B 0,C 180,E1 -13711.703,E2 -13711.703} C_VEL
LIN {X 0,Y 347.752,Z 243.669,A -85,B 0,C 180,E1 -13714.468,E2 -13714.468} C_VEL
LIN {X 0,Y 347.772,Z 243.657,A -85,B 0,C 180,E1 -13717.989,E2 -13717.989} C_VEL
LIN {X 0,Y 347.759,Z 243.659,A -85,B 0,C 180,E1 -13721.834,E2 -13721.834} C_VEL
LIN {X 0,Y 347.714,Z 243.638,A -85,B 0,C 180,E1 -13725.03,E2 -13725.03} C_VEL
LIN {X 0,Y 347.753,Z 243.664,A -85,B 0,C 180,E1 -13728.402,E2 -13728.402} C_VEL
LIN {X 0,Y 347.768,Z 243.659,A -85,B 0,C 180,E1 -13732.681,E2 -13732.681} C_VEL
LIN {X 0,Y 347.761,Z 243.661,A -85,B 0,C 180,E1 -13735.958,E2 -13735.958} C_VEL
LIN {X 0,Y 347.755,Z 243.67,A -85,B 0,C 180,E1 -13739.653,E2 -13739.653} C_VEL
LIN {X 0,Y 347.883,Z 243.754,A -85,B 0,C 180,E1 -13741.493,E2 -13741.493} C_VEL
LIN {X 0,Y 349.779,Z 253.72,A -85,B 0,C 180,E1 -13744.273,E2 -13744.273} C_VEL
LIN {X 0,Y 350.878,Z 260.489,A -85,B 0,C 180,E1 -13746.072,E2 -13746.072} C_VEL
LIN {X 0,Y 350.264,Z 268.296,A -85,B 0,C 180,E1 -13747.98,E2 -13747.98} C_VEL
LIN {X 0,Y 350.775,Z 272.306,A -85,B 0,C 180,E1 -13748.16,E2 -13748.16} C_VEL
LIN {X 0,Y 355.172,Z 301.436,A -85,B 0,C 180,E1 -13749.004,E2 -13749.004} C_VEL
LIN {X 0,Y 353.902,Z 376.12,A -85,B 0,C 180,E1 -13750.534,E2 -13750.534} C_VEL
LIN {X 0,Y 353.306,Z 389.425,A -85,B 0,C 180,E1 -13751.028,E2 -13751.028} C_VEL
LIN {X 0,Y 352.432,Z 402.754,A -85,B 0,C 180,E1 -13751.771,E2 -13751.771} C_VEL
LIN {X 0,Y 351.475,Z 414.741,A -85,B 0,C 180,E1 -13752.697,E2 -13752.697} C_VEL
LIN {X 0,Y 350.62,Z 424.941,A -85,B 0,C 180,E1 -13753.703,E2 -13753.703} C_VEL
LIN {X 0,Y 349.703,Z 435.538,A -85,B 0,C 180,E1 -13755.005,E2 -13755.005} C_VEL
LIN {X 0,Y 348.778,Z 444.174,A -85,B 0,C 180,E1 -13756.305,E2 -13756.305} C_VEL
LIN {X 0,Y 347.972,Z 452.129,A -85,B 0,C 180,E1 -13757.757,E2 -13757.757} C_VEL
LIN {X 0,Y 347.247,Z 459.881,A -85,B 0,C 180,E1 -13759.505,E2 -13759.505} C_VEL
LIN {X 0,Y 346.712,Z 466.092,A -85,B 0,C 180,E1 -13761.256,E2 -13761.256} C_VEL
LIN {X 0,Y 346.356,Z 471.012,A -85,B 0,C 180,E1 -13763.007,E2 -13763.007} C_VEL
LIN {X 0,Y 346.183,Z 474.394,A -85,B 0,C 180,E1 -13764.544,E2 -13764.544} C_VEL
LIN {X 0,Y 346.131,Z 477.534,A -85,B 0,C 180,E1 -13766.508,E2 -13766.508} C_VEL
LIN {X 0,Y 346.058,Z 479.719,A -85,B 0,C 180,E1 -13768.837,E2 -13768.837} C_VEL
LIN {X 0,Y 346.084,Z 480.191,A -85,B 0,C 180,E1 -13770,E2 -13770} C_VEL
LIN {X 0,Y 346.057,Z 480.249,A -85,B 0,C 180,E1 -13771.164,E2 -13771.164} C_VEL
LIN {X 0,Y 346.137,Z 479.217,A -85,B 0,C 180,E1 -13773.493,E2 -13773.493} C_VEL
LIN {X 0,Y 346.22,Z 478.099,A -85,B 0,C 180,E1 -13774.658,E2 -13774.658} C_VEL
LIN {X 0,Y 346.443,Z 474.58,A -85,B 0,C 180,E1 -13776.992,E2 -13776.992} C_VEL
LIN {X 0,Y 346.886,Z 470.785,A -85,B 0,C 180,E1 -13778.74,E2 -13778.74} C_VEL
LIN {X 0,Y 347.552,Z 465.889,A -85,B 0,C 180,E1 -13780.486,E2 -13780.486} C_VEL
LIN {X 0,Y 348.392,Z 459.744,A -85,B 0,C 180,E1 -13782.229,E2 -13782.229} C_VEL
LIN {X 0,Y 349.606,Z 452.114,A -85,B 0,C 180,E1 -13783.96,E2 -13783.96} C_VEL
LIN {X 0,Y 350.894,Z 443.379,A -85,B 0,C 180,E1 -13785.549,E2 -13785.549} C_VEL
LIN {X 0,Y 352.232,Z 432.942,A -85,B 0,C 180,E1 -13787.086,E2 -13787.086} C_VEL
LIN {X 0,Y 353.808,Z 421.686,A -85,B 0,C 180,E1 -13788.382,E2 -13788.382} C_VEL
LIN {X 0,Y 355.123,Z 410.899,A -85,B 0,C 180,E1 -13789.359,E2 -13789.359} C_VEL
LIN {X 0,Y 356.299,Z 399.032,A -85,B 0,C 180,E1 -13790.194,E2 -13790.194} C_VEL
LIN {X 0,Y 357.221,Z 386.995,A -85,B 0,C 180,E1 -13790.816,E2 -13790.816} C_VEL
LIN {X 0,Y 357.905,Z 373.565,A -85,B 0,C 180,E1 -13791.264,E2 -13791.264} C_VEL
LIN {X 0,Y 359.415,Z 302.042,A -85,B 0,C 180,E1 -13792.751,E2 -13792.751} C_VEL
LIN {X 0,Y 355.999,Z 283.61,A -85,B 0,C 180,E1 -13793.448,E2 -13793.448} C_VEL
LIN {X 0,Y 352.489,Z 268.142,A -85,B 0,C 180,E1 -13794.143,E2 -13794.143} C_VEL
LIN {X 0,Y 352.344,Z 264.481,A -85,B 0,C 180,E1 -13795.059,E2 -13795.059} C_VEL
LIN {X 0,Y 350.317,Z 254.243,A -85,B 0,C 180,E1 -13798.022,E2 -13798.022} C_VEL
LIN {X 0,Y 347.798,Z 243.833,A -85,B 0,C 180,E1 -13801.27,E2 -13801.27} C_VEL
LIN {X 0,Y 347.759,Z 243.667,A -85,B 0,C 180,E1 -13804.462,E2 -13804.462} C_VEL
LIN {X 0,Y 347.777,Z 243.659,A -85,B 0,C 180,E1 -13807.984,E2 -13807.984} C_VEL
LIN {X 0,Y 347.758,Z 243.658,A -85,B 0,C 180,E1 -13811.829,E2 -13811.829} C_VEL
LIN {X 0,Y 347.719,Z 243.672,A -85,B 0,C 180,E1 -13815.025,E2 -13815.025} C_VEL
LIN {X 0,Y 347.763,Z 243.652,A -85,B 0,C 180,E1 -13818.395,E2 -13818.395} C_VEL
LIN {X 0,Y 347.776,Z 243.66,A -85,B 0,C 180,E1 -13822.011,E2 -13822.011} C_VEL
LIN {X 0,Y 347.755,Z 243.666,A -85,B 0,C 180,E1 -13825.533,E2 -13825.533} C_VEL
LIN {X 0,Y 347.754,Z 243.66,A -85,B 0,C 180,E1 -13828.297,E2 -13828.297} C_VEL
LIN {X 0,Y 347.755,Z 243.663,A -85,B 0,C 180,E1 -13830.981,E2 -13830.981} C_VEL
LIN {X 0,Y 347.751,Z 243.667,A -85,B 0,C 180,E1 -13833.597,E2 -13833.597} C_VEL
LIN {X 0,Y 347.762,Z 243.658,A -85,B 0,C 180,E1 -13836.155,E2 -13836.155} C_VEL
LIN {X 0,Y 347.807,Z 243.651,A -85,B 0,C 180,E1 -13839.904,E2 -13839.904} C_VEL
LIN {X 0,Y 347.84,Z 243.65,A -85,B 0,C 180,E1 -13843.564,E2 -13843.564} C_VEL
LIN {X 0,Y 347.897,Z 243.649,A -85,B 0,C 180,E1 -13847.156,E2 -13847.156} C_VEL
LIN {X 0,Y 347.941,Z 243.641,A -85,B 0,C 180,E1 -13850.696,E2 -13850.696} C_VEL
LIN {X 0,Y 348.077,Z 243.622,A -85,B 0,C 180,E1 -13853.037,E2 -13853.037} C_VEL
LIN {X 0,Y 348.196,Z 243.607,A -85,B 0,C 180,E1 -13857.681,E2 -13857.681} C_VEL
LIN {X 0,Y 348.303,Z 243.596,A -85,B 0,C 180,E1 -13859.995,E2 -13859.995} C_VEL
LIN {X 0,Y 348.196,Z 243.604,A -85,B 0,C 180,E1 -13862.308,E2 -13862.308} C_VEL
LIN {X 0,Y 348.067,Z 243.618,A -85,B 0,C 180,E1 -13866.953,E2 -13866.953} C_VEL
LIN {X 0,Y 347.921,Z 243.642,A -85,B 0,C 180,E1 -13870.469,E2 -13870.469} C_VEL
LIN {X 0,Y 347.891,Z 243.651,A -85,B 0,C 180,E1 -13874.144,E2 -13874.144} C_VEL
LIN {X 0,Y 347.819,Z 243.657,A -85,B 0,C 180,E1 -13878.253,E2 -13878.253} C_VEL
LIN {X 0,Y 347.776,Z 243.658,A -85,B 0,C 180,E1 -13881.629,E2 -13881.629} C_VEL
LIN {X 0,Y 347.797,Z 243.649,A -85,B 0,C 180,E1 -13885.103,E2 -13885.103} C_VEL
LIN {X 0,Y 347.791,Z 243.656,A -85,B 0,C 180,E1 -13887.688,E2 -13887.688} C_VEL
LIN {X 0,Y 347.73,Z 243.66,A -85,B 0,C 180,E1 -13890.342,E2 -13890.342} C_VEL
LIN {X 0,Y 347.726,Z 243.667,A -85,B 0,C 180,E1 -13894.038,E2 -13894.038} C_VEL
LIN {X 0,Y 347.745,Z 243.666,A -85,B 0,C 180,E1 -13897.314,E2 -13897.314} C_VEL
LIN {X 0,Y 347.768,Z 243.663,A -85,B 0,C 180,E1 -13900.283,E2 -13900.283} C_VEL
LIN {X 0,Y 347.811,Z 243.777,A -85,B 0,C 180,E1 -13902.988,E2 -13902.988} C_VEL
LIN {X 0,Y 349.78,Z 252.113,A -85,B 0,C 180,E1 -13905.636,E2 -13905.636} C_VEL
LIN {X 0,Y 351.375,Z 259.564,A -85,B 0,C 180,E1 -13907.787,E2 -13907.787} C_VEL
LIN {X 0,Y 354.504,Z 267.141,A -85,B 0,C 180,E1 -13908.285,E2 -13908.285} C_VEL
LIN {X 0,Y 357.918,Z 280.782,A -85,B 0,C 180,E1 -13908.886,E2 -13908.886} C_VEL
LIN {X 0,Y 359.743,Z 290.109,A -85,B 0,C 180,E1 -13909.245,E2 -13909.245} C_VEL
LIN {X 0,Y 357.936,Z 367.106,A -85,B 0,C 180,E1 -13910.848,E2 -13910.848} C_VEL
LIN {X 0,Y 357.196,Z 380.769,A -85,B 0,C 180,E1 -13911.362,E2 -13911.362} C_VEL
LIN {X 0,Y 356.17,Z 393.917,A -85,B 0,C 180,E1 -13912.107,E2 -13912.107} C_VEL
LIN {X 0,Y 354.94,Z 405.749,A -85,B 0,C 180,E1 -13913.027,E2 -13913.027} C_VEL
LIN {X 0,Y 353.684,Z 416.602,A -85,B 0,C 180,E1 -13914.113,E2 -13914.113} C_VEL
LIN {X 0,Y 352.351,Z 426.583,A -85,B 0,C 180,E1 -13915.357,E2 -13915.357} C_VEL
LIN {X 0,Y 350.874,Z 436.613,A -85,B 0,C 180,E1 -13916.919,E2 -13916.919} C_VEL
LIN {X 0,Y 349.647,Z 444.732,A -85,B 0,C 180,E1 -13918.492,E2 -13918.492} C_VEL
LIN {X 0,Y 348.554,Z 451.498,A -85,B 0,C 180,E1 -13920.099,E2 -13920.099} C_VEL
LIN {X 0,Y 347.777,Z 456.8,A -85,B 0,C 180,E1 -13921.647,E2 -13921.647} C_VEL
LIN {X 0,Y 347.053,Z 461.963,A -85,B 0,C 180,E1 -13923.544,E2 -13923.544} C_VEL
LIN {X 0,Y 346.699,Z 464.688,A -85,B 0,C 180,E1 -13924.805,E2 -13924.805} C_VEL
LIN {X 0,Y 346.432,Z 466.836,A -85,B 0,C 180,E1 -13926.062,E2 -13926.062} C_VEL
LIN {X 0,Y 346.173,Z 468.515,A -85,B 0,C 180,E1 -13927.31,E2 -13927.31} C_VEL
LIN {X 0,Y 346.014,Z 470.07,A -85,B 0,C 180,E1 -13929.097,E2 -13929.097} C_VEL
LIN {X 0,Y 345.883,Z 470.712,A -85,B 0,C 180,E1 -13931.028,E2 -13931.028} C_VEL
LIN {X 0,Y 345.905,Z 470.372,A -85,B 0,C 180,E1 -13932.707,E2 -13932.707} C_VEL
LIN {X 0,Y 345.919,Z 468.926,A -85,B 0,C 180,E1 -13934.685,E2 -13934.685} C_VEL
LIN {X 0,Y 346.026,Z 467.479,A -85,B 0,C 180,E1 -13935.893,E2 -13935.893} C_VEL
LIN {X 0,Y 346.315,Z 464.424,A -85,B 0,C 180,E1 -13937.697,E2 -13937.697} C_VEL
LIN {X 0,Y 346.57,Z 460.298,A -85,B 0,C 180,E1 -13939.484,E2 -13939.484} C_VEL
LIN {X 0,Y 347.136,Z 453.931,A -85,B 0,C 180,E1 -13941.559,E2 -13941.559} C_VEL
LIN {X 0,Y 347.79,Z 447.005,A -85,B 0,C 180,E1 -13943.327,E2 -13943.327} C_VEL
LIN {X 0,Y 348.456,Z 439.941,A -85,B 0,C 180,E1 -13944.792,E2 -13944.792} C_VEL
LIN {X 0,Y 349.257,Z 431.433,A -85,B 0,C 180,E1 -13946.25,E2 -13946.25} C_VEL
LIN {X 0,Y 350.32,Z 420.873,A -85,B 0,C 180,E1 -13947.7,E2 -13947.7} C_VEL
LIN {X 0,Y 351.408,Z 409.161,A -85,B 0,C 180,E1 -13948.978,E2 -13948.978} C_VEL
LIN {X 0,Y 352.364,Z 396.969,A -85,B 0,C 180,E1 -13950,E2 -13950} C_VEL
LIN {X 0,Y 353.092,Z 384.517,A -85,B 0,C 180,E1 -13950.784,E2 -13950.784} C_VEL
LIN {X 0,Y 353.704,Z 371.573,A -85,B 0,C 180,E1 -13951.352,E2 -13951.352} C_VEL
LIN {X 0,Y 354.119,Z 356.101,A -85,B 0,C 180,E1 -13951.741,E2 -13951.741} C_VEL
LIN {X 0,Y 355.197,Z 287.616,A -85,B 0,C 180,E1 -13953.134,E2 -13953.134} C_VEL
LIN {X 0,Y 350.478,Z 259.643,A -85,B 0,C 180,E1 -13954.008,E2 -13954.008} C_VEL
LIN {X 0,Y 350.341,Z 257.163,A -85,B 0,C 180,E1 -13954.602,E2 -13954.602} C_VEL
LIN {X 0,Y 348.625,Z 246.705,A -85,B 0,C 180,E1 -13957.529,E2 -13957.529} C_VEL
LIN {X 0,Y 348.031,Z 243.67,A -85,B 0,C 180,E1 -13958.488,E2 -13958.488} C_VEL
LIN {X 0,Y 347.874,Z 243.651,A -85,B 0,C 180,E1 -13961.655,E2 -13961.655} C_VEL
LIN {X 0,Y 347.877,Z 243.651,A -85,B 0,C 180,E1 -13963.095,E2 -13963.095} C_VEL
LIN {X 0,Y 347.226,Z 243.732,A -85,B 0,C 180,E1 -13964.06,E2 -13964.06} C_VEL
LIN {X 0,Y 344.394,Z 244.084,A -85,B 0,C 180,E1 -13965.63,E2 -13965.63} C_VEL
LIN {X 0,Y 341.971,Z 244.386,A -85,B 0,C 180,E1 -13966.901,E2 -13966.901} C_VEL
LIN {X 0,Y 340.91,Z 244.511,A -85,B 0,C 180,E1 -13967.885,E2 -13967.885} C_VEL
LIN {X 0,Y 340.812,Z 244.518,A -85,B 0,C 180,E1 -13968.218,E2 -13968.218} C_VEL
LIN {X 0,Y 340.769,Z 244.535,A -85,B 0,C 180,E1 -13971.884,E2 -13971.884} C_VEL
LIN {X 0,Y 340.734,Z 244.516,A -85,B 0,C 180,E1 -13975.667,E2 -13975.667} C_VEL
LIN {X 0,Y 340.709,Z 244.523,A -85,B 0,C 180,E1 -13978.322,E2 -13978.322} C_VEL
LIN {X 0,Y 340.719,Z 244.542,A -85,B 0,C 180,E1 -13981.042,E2 -13981.042} C_VEL
LIN {X 0,Y 340.716,Z 244.533,A -85,B 0,C 180,E1 -13985.278,E2 -13985.278} C_VEL
LIN {X 0,Y 340.744,Z 244.538,A -85,B 0,C 180,E1 -13988.405,E2 -13988.405} C_VEL
LIN {X 0,Y 340.747,Z 244.522,A -85,B 0,C 180,E1 -13992.065,E2 -13992.065} C_VEL
LIN {X 0,Y 340.762,Z 244.534,A -85,B 0,C 180,E1 -13995.484,E2 -13995.484} C_VEL
LIN {X 0,Y 340.697,Z 244.538,A -85,B 0,C 180,E1 -13998.702,E2 -13998.702} C_VEL
LIN {X 0,Y 340.713,Z 244.519,A -85,B 0,C 180,E1 -14001.779,E2 -14001.779} C_VEL
LIN {X 0,Y 340.697,Z 244.542,A -85,B 0,C 180,E1 -14005.601,E2 -14005.601} C_VEL
LIN {X 0,Y 340.692,Z 244.537,A -85,B 0,C 180,E1 -14008.963,E2 -14008.963} C_VEL
LIN {X 0,Y 340.759,Z 244.508,A -85,B 0,C 180,E1 -14012.479,E2 -14012.479} C_VEL
LIN {X 0,Y 340.745,Z 244.531,A -85,B 0,C 180,E1 -14015.645,E2 -14015.645} C_VEL
LIN {X 0,Y 340.761,Z 244.534,A -85,B 0,C 180,E1 -14019.482,E2 -14019.482} C_VEL
LIN {X 0,Y 340.844,Z 244.513,A -85,B 0,C 180,E1 -14021.99,E2 -14021.99} C_VEL
LIN {X 0,Y 340.857,Z 244.496,A -85,B 0,C 180,E1 -14025.711,E2 -14025.711} C_VEL
LIN {X 0,Y 340.866,Z 244.521,A -85,B 0,C 180,E1 -14029.312,E2 -14029.312} C_VEL
LIN {X 0,Y 341.069,Z 244.497,A -85,B 0,C 180,E1 -14032.904,E2 -14032.904} C_VEL
LIN {X 0,Y 341.163,Z 244.453,A -85,B 0,C 180,E1 -14037.644,E2 -14037.644} C_VEL
LIN {X 0,Y 341.272,Z 244.455,A -85,B 0,C 180,E1 -14040.005,E2 -14040.005} C_VEL
LIN {X 0,Y 341.165,Z 244.484,A -85,B 0,C 180,E1 -14042.366,E2 -14042.366} C_VEL
LIN {X 0,Y 341.016,Z 244.497,A -85,B 0,C 180,E1 -14047.108,E2 -14047.108} C_VEL
LIN {X 0,Y 340.85,Z 244.499,A -85,B 0,C 180,E1 -14050.699,E2 -14050.699} C_VEL
LIN {X 0,Y 340.867,Z 244.523,A -85,B 0,C 180,E1 -14054.329,E2 -14054.329} C_VEL
LIN {X 0,Y 340.842,Z 244.519,A -85,B 0,C 180,E1 -14058.471,E2 -14058.471} C_VEL
LIN {X 0,Y 340.724,Z 244.522,A -85,B 0,C 180,E1 -14061.846,E2 -14061.846} C_VEL
LIN {X 0,Y 340.779,Z 244.535,A -85,B 0,C 180,E1 -14065.668,E2 -14065.668} C_VEL
LIN {X 0,Y 340.727,Z 244.537,A -85,B 0,C 180,E1 -14068.325,E2 -14068.325} C_VEL
LIN {X 0,Y 340.703,Z 244.535,A -85,B 0,C 180,E1 -14071.049,E2 -14071.049} C_VEL
LIN {X 0,Y 340.725,Z 244.54,A -85,B 0,C 180,E1 -14075.283,E2 -14075.283} C_VEL
LIN {X 0,Y 340.703,Z 244.538,A -85,B 0,C 180,E1 -14078.386,E2 -14078.386} C_VEL
LIN {X 0,Y 340.708,Z 244.536,A -85,B 0,C 180,E1 -14082.048,E2 -14082.048} C_VEL
LIN {X 0,Y 340.662,Z 244.523,A -85,B 0,C 180,E1 -14086.23,E2 -14086.23} C_VEL
LIN {X 0,Y 340.683,Z 244.545,A -85,B 0,C 180,E1 -14088.691,E2 -14088.691} C_VEL
LIN {X 0,Y 340.73,Z 244.532,A -85,B 0,C 180,E1 -14091.773,E2 -14091.773} C_VEL
LIN {X 0,Y 340.736,Z 244.537,A -85,B 0,C 180,E1 -14095.598,E2 -14095.598} C_VEL
LIN {X 0,Y 340.707,Z 244.543,A -85,B 0,C 180,E1 -14098.957,E2 -14098.957} C_VEL
LIN {X 0,Y 340.798,Z 244.586,A -85,B 0,C 180,E1 -14101.182,E2 -14101.182} C_VEL
LIN {X 0,Y 341.536,Z 248.016,A -85,B 0,C 180,E1 -14102.238,E2 -14102.238} C_VEL
LIN {X 0,Y 343.751,Z 260.037,A -85,B 0,C 180,E1 -14105.543,E2 -14105.543} C_VEL
LIN {X 0,Y 343.749,Z 263.989,A -85,B 0,C 180,E1 -14106.569,E2 -14106.569} C_VEL
LIN {X 0,Y 343.381,Z 268.503,A -85,B 0,C 180,E1 -14107.644,E2 -14107.644} C_VEL
LIN {X 0,Y 348.39,Z 302.323,A -85,B 0,C 180,E1 -14108.677,E2 -14108.677} C_VEL
LIN {X 0,Y 347.092,Z 375.747,A -85,B 0,C 180,E1 -14110.213,E2 -14110.213} C_VEL
LIN {X 0,Y 346.525,Z 388.391,A -85,B 0,C 180,E1 -14110.681,E2 -14110.681} C_VEL
LIN {X 0,Y 345.665,Z 401.409,A -85,B 0,C 180,E1 -14111.401,E2 -14111.401} C_VEL
LIN {X 0,Y 344.642,Z 413.763,A -85,B 0,C 180,E1 -14112.343,E2 -14112.343} C_VEL
LIN {X 0,Y 343.641,Z 425.437,A -85,B 0,C 180,E1 -14113.516,E2 -14113.516} C_VEL
LIN {X 0,Y 342.698,Z 435.938,A -85,B 0,C 180,E1 -14114.843,E2 -14114.843} C_VEL
LIN {X 0,Y 341.678,Z 445.344,A -85,B 0,C 180,E1 -14116.318,E2 -14116.318} C_VEL
LIN {X 0,Y 340.659,Z 454.43,A -85,B 0,C 180,E1 -14118.095,E2 -14118.095} C_VEL
LIN {X 0,Y 340.002,Z 461.744,A -85,B 0,C 180,E1 -14119.881,E2 -14119.881} C_VEL
LIN {X 0,Y 339.533,Z 467.577,A -85,B 0,C 180,E1 -14121.669,E2 -14121.669} C_VEL
LIN {X 0,Y 339.217,Z 472.152,A -85,B 0,C 180,E1 -14123.457,E2 -14123.457} C_VEL
LIN {X 0,Y 339.075,Z 475.619,A -85,B 0,C 180,E1 -14125.245,E2 -14125.245} C_VEL
LIN {X 0,Y 339.057,Z 477.344,A -85,B 0,C 180,E1 -14126.435,E2 -14126.435} C_VEL
LIN {X 0,Y 338.964,Z 479.569,A -85,B 0,C 180,E1 -14128.812,E2 -14128.812} C_VEL
LIN {X 0,Y 338.987,Z 480.08,A -85,B 0,C 180,E1 -14130,E2 -14130} C_VEL
LIN {X 0,Y 338.963,Z 480.16,A -85,B 0,C 180,E1 -14131.188,E2 -14131.188} C_VEL
LIN {X 0,Y 339.066,Z 479.17,A -85,B 0,C 180,E1 -14133.565,E2 -14133.565} C_VEL
LIN {X 0,Y 339.121,Z 478.09,A -85,B 0,C 180,E1 -14134.755,E2 -14134.755} C_VEL
LIN {X 0,Y 339.185,Z 476.564,A -85,B 0,C 180,E1 -14135.947,E2 -14135.947} C_VEL
LIN {X 0,Y 339.513,Z 473.506,A -85,B 0,C 180,E1 -14137.733,E2 -14137.733} C_VEL
LIN {X 0,Y 340.069,Z 469.409,A -85,B 0,C 180,E1 -14139.517,E2 -14139.517} C_VEL
LIN {X 0,Y 341.006,Z 463.159,A -85,B 0,C 180,E1 -14141.592,E2 -14141.592} C_VEL
LIN {X 0,Y 342.009,Z 456.374,A -85,B 0,C 180,E1 -14143.367,E2 -14143.367} C_VEL
LIN {X 0,Y 343.439,Z 447.937,A -85,B 0,C 180,E1 -14145.124,E2 -14145.124} C_VEL
LIN {X 0,Y 344.632,Z 439.294,A -85,B 0,C 180,E1 -14146.589,E2 -14146.589} C_VEL
LIN {X 0,Y 346.189,Z 428.669,A -85,B 0,C 180,E1 -14148.035,E2 -14148.035} C_VEL
LIN {X 0,Y 347.651,Z 418.113,A -85,B 0,C 180,E1 -14149.178,E2 -14149.178} C_VEL
LIN {X 0,Y 349.035,Z 406.357,A -85,B 0,C 180,E1 -14150.171,E2 -14150.171} C_VEL
LIN {X 0,Y 350.3,Z 392.91,A -85,B 0,C 180,E1 -14151.016,E2 -14151.016} C_VEL
LIN {X 0,Y 351.228,Z 379.771,A -85,B 0,C 180,E1 -14151.573,E2 -14151.573} C_VEL
LIN {X 0,Y 351.79,Z 362.465,A -85,B 0,C 180,E1 -14151.999,E2 -14151.999} C_VEL
LIN {X 0,Y 353.087,Z 303.158,A -85,B 0,C 180,E1 -14153.246,E2 -14153.246} C_VEL
LIN {X 0,Y 349.86,Z 285.631,A -85,B 0,C 180,E1 -14153.927,E2 -14153.927} C_VEL
LIN {X 0,Y 345.82,Z 268.531,A -85,B 0,C 180,E1 -14154.707,E2 -14154.707} C_VEL
LIN {X 0,Y 345.625,Z 267.068,A -85,B 0,C 180,E1 -14154.957,E2 -14154.957} C_VEL
LIN {X 0,Y 343.842,Z 257.686,A -85,B 0,C 180,E1 -14157.711,E2 -14157.711} C_VEL
LIN {X 0,Y 341.381,Z 247.243,A -85,B 0,C 180,E1 -14160.976,E2 -14160.976} C_VEL
LIN {X 0,Y 340.723,Z 244.597,A -85,B 0,C 180,E1 -14161.924,E2 -14161.924} C_VEL
LIN {X 0,Y 340.732,Z 244.535,A -85,B 0,C 180,E1 -14165.277,E2 -14165.277} C_VEL
LIN {X 0,Y 340.708,Z 244.536,A -85,B 0,C 180,E1 -14168.38,E2 -14168.38} C_VEL
LIN {X 0,Y 340.708,Z 244.534,A -85,B 0,C 180,E1 -14172.042,E2 -14172.042} C_VEL
LIN {X 0,Y 340.666,Z 244.538,A -85,B 0,C 180,E1 -14176.225,E2 -14176.225} C_VEL
LIN {X 0,Y 340.69,Z 244.546,A -85,B 0,C 180,E1 -14179.753,E2 -14179.753} C_VEL
LIN {X 0,Y 340.714,Z 244.544,A -85,B 0,C 180,E1 -14183.255,E2 -14183.255} C_VEL
LIN {X 0,Y 340.705,Z 244.545,A -85,B 0,C 180,E1 -14186.15,E2 -14186.15} C_VEL
LIN {X 0,Y 340.73,Z 244.541,A -85,B 0,C 180,E1 -14190.032,E2 -14190.032} C_VEL
LIN {X 0,Y 340.726,Z 244.54,A -85,B 0,C 180,E1 -14193.009,E2 -14193.009} C_VEL
LIN {X 0,Y 340.715,Z 244.539,A -85,B 0,C 180,E1 -14196.922,E2 -14196.922} C_VEL
LIN {X 0,Y 340.743,Z 244.532,A -85,B 0,C 180,E1 -14200.726,E2 -14200.726} C_VEL
LIN {X 0,Y 340.825,Z 244.518,A -85,B 0,C 180,E1 -14204.446,E2 -14204.446} C_VEL
LIN {X 0,Y 340.856,Z 244.52,A -85,B 0,C 180,E1 -14208.096,E2 -14208.096} C_VEL
LIN {X 0,Y 340.985,Z 244.513,A -85,B 0,C 180,E1 -14211.7,E2 -14211.7} C_VEL
LIN {X 0,Y 341.03,Z 244.496,A -85,B 0,C 180,E1 -14214.081,E2 -14214.081} C_VEL
LIN {X 0,Y 341.133,Z 244.487,A -85,B 0,C 180,E1 -14217.633,E2 -14217.633} C_VEL
LIN {X 0,Y 341.255,Z 244.474,A -85,B 0,C 180,E1 -14219.995,E2 -14219.995} C_VEL
LIN {X 0,Y 341.157,Z 244.48,A -85,B 0,C 180,E1 -14222.356,E2 -14222.356} C_VEL
LIN {X 0,Y 341.015,Z 244.496,A -85,B 0,C 180,E1 -14227.097,E2 -14227.097} C_VEL
LIN {X 0,Y 340.864,Z 244.519,A -85,B 0,C 180,E1 -14230.688,E2 -14230.688} C_VEL
LIN {X 0,Y 340.856,Z 244.525,A -85,B 0,C 180,E1 -14234.319,E2 -14234.319} C_VEL
LIN {X 0,Y 340.776,Z 244.533,A -85,B 0,C 180,E1 -14238.435,E2 -14238.435} C_VEL
LIN {X 0,Y 340.741,Z 244.535,A -85,B 0,C 180,E1 -14241.851,E2 -14241.851} C_VEL
LIN {X 0,Y 340.756,Z 244.52,A -85,B 0,C 180,E1 -14245.658,E2 -14245.658} C_VEL
LIN {X 0,Y 340.711,Z 244.543,A -85,B 0,C 180,E1 -14248.315,E2 -14248.315} C_VEL
LIN {X 0,Y 340.678,Z 244.535,A -85,B 0,C 180,E1 -14251.039,E2 -14251.039} C_VEL
LIN {X 0,Y 340.696,Z 244.537,A -85,B 0,C 180,E1 -14255.273,E2 -14255.273} C_VEL
LIN {X 0,Y 340.701,Z 244.537,A -85,B 0,C 180,E1 -14258.384,E2 -14258.384} C_VEL
LIN {X 0,Y 340.746,Z 244.543,A -85,B 0,C 180,E1 -14262.158,E2 -14262.158} C_VEL
LIN {X 0,Y 340.802,Z 244.841,A -85,B 0,C 180,E1 -14262.522,E2 -14262.522} C_VEL
LIN {X 0,Y 343.179,Z 255.001,A -85,B 0,C 180,E1 -14265.778,E2 -14265.778} C_VEL
LIN {X 0,Y 344.203,Z 259.677,A -85,B 0,C 180,E1 -14267.139,E2 -14267.139} C_VEL
LIN {X 0,Y 348.932,Z 270.83,A -85,B 0,C 180,E1 -14267.883,E2 -14267.883} C_VEL
LIN {X 0,Y 352.636,Z 287.03,A -85,B 0,C 180,E1 -14268.581,E2 -14268.581} C_VEL
LIN {X 0,Y 353.392,Z 290.974,A -85,B 0,C 180,E1 -14268.736,E2 -14268.736} C_VEL
LIN {X 0,Y 351.522,Z 367.496,A -85,B 0,C 180,E1 -14270.364,E2 -14270.364} C_VEL
LIN {X 0,Y 350.731,Z 381.02,A -85,B 0,C 180,E1 -14270.884,E2 -14270.884} C_VEL
LIN {X 0,Y 349.746,Z 393.315,A -85,B 0,C 180,E1 -14271.588,E2 -14271.588} C_VEL
LIN {X 0,Y 348.405,Z 405.912,A -85,B 0,C 180,E1 -14272.578,E2 -14272.578} C_VEL
LIN {X 0,Y 347.068,Z 416.725,A -85,B 0,C 180,E1 -14273.679,E2 -14273.679} C_VEL
LIN {X 0,Y 345.657,Z 426.895,A -85,B 0,C 180,E1 -14274.972,E2 -14274.972} C_VEL
LIN {X 0,Y 344.127,Z 436.731,A -85,B 0,C 180,E1 -14276.536,E2 -14276.536} C_VEL
LIN {X 0,Y 342.827,Z 444.844,A -85,B 0,C 180,E1 -14278.138,E2 -14278.138} C_VEL
LIN {X 0,Y 341.508,Z 452.669,A -85,B 0,C 180,E1 -14280.059,E2 -14280.059} C_VEL
LIN {X 0,Y 340.673,Z 457.88,A -85,B 0,C 180,E1 -14281.674,E2 -14281.674} C_VEL
LIN {X 0,Y 339.944,Z 462.82,A -85,B 0,C 180,E1 -14283.609,E2 -14283.609} C_VEL
LIN {X 0,Y 339.421,Z 466.606,A -85,B 0,C 180,E1 -14285.633,E2 -14285.633} C_VEL
LIN {X 0,Y 339.173,Z 468.234,A -85,B 0,C 180,E1 -14286.815,E2 -14286.815} C_VEL
LIN {X 0,Y 338.947,Z 470.13,A -85,B 0,C 180,E1 -14288.896,E2 -14288.896} C_VEL
LIN {X 0,Y 338.793,Z 470.771,A -85,B 0,C 180,E1 -14290.615,E2 -14290.615} C_VEL
LIN {X 0,Y 338.805,Z 470.503,A -85,B 0,C 180,E1 -14292.566,E2 -14292.566} C_VEL
LIN {X 0,Y 338.802,Z 469.318,A -85,B 0,C 180,E1 -14294.355,E2 -14294.355} C_VEL
LIN {X 0,Y 338.898,Z 467.963,A -85,B 0,C 180,E1 -14295.59,E2 -14295.59} C_VEL
LIN {X 0,Y 339.207,Z 465.006,A -85,B 0,C 180,E1 -14297.474,E2 -14297.474} C_VEL
LIN {X 0,Y 339.44,Z 461.139,A -85,B 0,C 180,E1 -14299.26,E2 -14299.26} C_VEL
LIN {X 0,Y 339.866,Z 456.03,A -85,B 0,C 180,E1 -14301.078,E2 -14301.078} C_VEL
LIN {X 0,Y 340.52,Z 449.589,A -85,B 0,C 180,E1 -14302.886,E2 -14302.886} C_VEL
LIN {X 0,Y 341.316,Z 441.52,A -85,B 0,C 180,E1 -14304.683,E2 -14304.683} C_VEL
LIN {X 0,Y 342.077,Z 433.312,A -85,B 0,C 180,E1 -14306.171,E2 -14306.171} C_VEL
LIN {X 0,Y 343.154,Z 423.255,A -85,B 0,C 180,E1 -14307.652,E2 -14307.652} C_VEL
LIN {X 0,Y 344.291,Z 412.103,A -85,B 0,C 180,E1 -14308.951,E2 -14308.951} C_VEL
LIN {X 0,Y 345.217,Z 400.721,A -85,B 0,C 180,E1 -14310,E2 -14310} C_VEL
LIN {X 0,Y 346.071,Z 388.347,A -85,B 0,C 180,E1 -14310.872,E2 -14310.872} C_VEL
LIN {X 0,Y 346.683,Z 376.135,A -85,B 0,C 180,E1 -14311.488,E2 -14311.488} C_VEL
LIN {X 0,Y 347.166,Z 362.605,A -85,B 0,C 180,E1 -14311.921,E2 -14311.921} C_VEL
LIN {X 0,Y 348.484,Z 288.837,A -85,B 0,C 180,E1 -14313.45,E2 -14313.45} C_VEL
LIN {X 0,Y 343.601,Z 260.058,A -85,B 0,C 180,E1 -14314.362,E2 -14314.362} C_VEL
LIN {X 0,Y 343.457,Z 258.938,A -85,B 0,C 180,E1 -14314.548,E2 -14314.548} C_VEL
LIN {X 0,Y 341.644,Z 247.948,A -85,B 0,C 180,E1 -14317.664,E2 -14317.664} C_VEL
LIN {X 0,Y 340.955,Z 244.58,A -85,B 0,C 180,E1 -14318.732,E2 -14318.732} C_VEL
LIN {X 0,Y 340.86,Z 244.527,A -85,B 0,C 180,E1 -14323.108,E2 -14323.108} C_VEL
LIN {X 0,Y 340.761,Z 244.538,A -85,B 0,C 180,E1 -14326.782,E2 -14326.782} C_VEL
LIN {X 0,Y 340.812,Z 244.518,A -85,B 0,C 180,E1 -14328.218,E2 -14328.218} C_VEL
LIN {X 0,Y 340.101,Z 244.601,A -85,B 0,C 180,E1 -14329.204,E2 -14329.204} C_VEL
LIN {X 0,Y 337.193,Z 244.971,A -85,B 0,C 180,E1 -14330.806,E2 -14330.806} C_VEL
LIN {X 0,Y 334.768,Z 245.282,A -85,B 0,C 180,E1 -14332.104,E2 -14332.104} C_VEL
LIN {X 0,Y 333.753,Z 245.411,A -85,B 0,C 180,E1 -14333.109,E2 -14333.109} C_VEL
LIN {X 0,Y 333.683,Z 245.415,A -85,B 0,C 180,E1 -14333.449,E2 -14333.449} C_VEL
LIN {X 0,Y 333.696,Z 245.386,A -85,B 0,C 180,E1 -14336.249,E2 -14336.249} C_VEL
LIN {X 0,Y 333.689,Z 245.4,A -85,B 0,C 180,E1 -14338.974,E2 -14338.974} C_VEL
LIN {X 0,Y 333.668,Z 245.422,A -85,B 0,C 180,E1 -14342.608,E2 -14342.608} C_VEL
LIN {X 0,Y 333.689,Z 245.413,A -85,B 0,C 180,E1 -14346.137,E2 -14346.137} C_VEL
LIN {X 0,Y 333.686,Z 245.419,A -85,B 0,C 180,E1 -14349.186,E2 -14349.186} C_VEL
LIN {X 0,Y 333.688,Z 245.4,A -85,B 0,C 180,E1 -14352.521,E2 -14352.521} C_VEL
LIN {X 0,Y 333.705,Z 245.419,A -85,B 0,C 180,E1 -14355.983,E2 -14355.983} C_VEL
LIN {X 0,Y 333.672,Z 245.412,A -85,B 0,C 180,E1 -14359.309,E2 -14359.309} C_VEL
LIN {X 0,Y 333.64,Z 245.411,A -85,B 0,C 180,E1 -14363.173,E2 -14363.173} C_VEL
LIN {X 0,Y 333.617,Z 245.427,A -85,B 0,C 180,E1 -14366.798,E2 -14366.798} C_VEL
LIN {X 0,Y 333.682,Z 245.409,A -85,B 0,C 180,E1 -14369.715,E2 -14369.715} C_VEL
LIN {X 0,Y 333.723,Z 245.383,A -85,B 0,C 180,E1 -14372.407,E2 -14372.407} C_VEL
LIN {X 0,Y 333.714,Z 245.406,A -85,B 0,C 180,E1 -14375.097,E2 -14375.097} C_VEL
LIN {X 0,Y 333.694,Z 245.418,A -85,B 0,C 180,E1 -14379.027,E2 -14379.027} C_VEL
LIN {X 0,Y 333.781,Z 245.393,A -85,B 0,C 180,E1 -14381.595,E2 -14381.595} C_VEL
LIN {X 0,Y 333.796,Z 245.373,A -85,B 0,C 180,E1 -14385.582,E2 -14385.582} C_VEL
LIN {X 0,Y 333.828,Z 245.394,A -85,B 0,C 180,E1 -14389.084,E2 -14389.084} C_VEL
LIN {X 0,Y 334.018,Z 245.374,A -85,B 0,C 180,E1 -14392.753,E2 -14392.753} C_VEL
LIN {X 0,Y 333.805,Z 245.388,A -85,B 0,C 180,E1 -14395.175,E2 -14395.175} C_VEL
LIN {X 0,Y 334.1,Z 245.332,A -85,B 0,C 180,E1 -14397.594,E2 -14397.594} C_VEL
LIN {X 0,Y 334.224,Z 245.332,A -85,B 0,C 180,E1 -14400.005,E2 -14400.005} C_VEL
LIN {X 0,Y 334.103,Z 245.364,A -85,B 0,C 180,E1 -14402.417,E2 -14402.417} C_VEL
LIN {X 0,Y 333.998,Z 245.376,A -85,B 0,C 180,E1 -14406.044,E2 -14406.044} C_VEL
LIN {X 0,Y 333.822,Z 245.373,A -85,B 0,C 180,E1 -14409.701,E2 -14409.701} C_VEL
LIN {X 0,Y 333.8,Z 245.395,A -85,B 0,C 180,E1 -14413.396,E2 -14413.396} C_VEL
LIN {X 0,Y 333.751,Z 245.407,A -85,B 0,C 180,E1 -14417.151,E2 -14417.151} C_VEL
LIN {X 0,Y 333.737,Z 245.398,A -85,B 0,C 180,E1 -14419.695,E2 -14419.695} C_VEL
LIN {X 0,Y 333.676,Z 245.414,A -85,B 0,C 180,E1 -14423.594,E2 -14423.594} C_VEL
LIN {X 0,Y 333.737,Z 245.414,A -85,B 0,C 180,E1 -14426.251,E2 -14426.251} C_VEL
LIN {X 0,Y 333.688,Z 245.404,A -85,B 0,C 180,E1 -14428.979,E2 -14428.979} C_VEL
LIN {X 0,Y 333.646,Z 245.429,A -85,B 0,C 180,E1 -14433.212,E2 -14433.212} C_VEL
LIN {X 0,Y 333.683,Z 245.413,A -85,B 0,C 180,E1 -14436.143,E2 -14436.143} C_VEL
LIN {X 0,Y 333.643,Z 245.423,A -85,B 0,C 180,E1 -14439.198,E2 -14439.198} C_VEL
LIN {X 0,Y 333.643,Z 245.416,A -85,B 0,C 180,E1 -14442.503,E2 -14442.503} C_VEL
LIN {X 0,Y 333.606,Z 245.398,A -85,B 0,C 180,E1 -14445.957,E2 -14445.957} C_VEL
LIN {X 0,Y 333.614,Z 245.429,A -85,B 0,C 180,E1 -14449.327,E2 -14449.327} C_VEL
LIN {X 0,Y 333.675,Z 245.416,A -85,B 0,C 180,E1 -14453.171,E2 -14453.171} C_VEL
LIN {X 0,Y 333.686,Z 245.416,A -85,B 0,C 180,E1 -14455.343,E2 -14455.343} C_VEL
LIN {X 0,Y 333.642,Z 245.422,A -85,B 0,C 180,E1 -14458.224,E2 -14458.224} C_VEL
LIN {X 0,Y 333.743,Z 245.529,A -85,B 0,C 180,E1 -14460.945,E2 -14460.945} C_VEL
LIN {X 0,Y 335.547,Z 254.506,A -85,B 0,C 180,E1 -14463.572,E2 -14463.572} C_VEL
LIN {X 0,Y 336.88,Z 262.051,A -85,B 0,C 180,E1 -14465.668,E2 -14465.668} C_VEL
LIN {X 0,Y 336.488,Z 268.368,A -85,B 0,C 180,E1 -14467.249,E2 -14467.249} C_VEL
LIN {X 0,Y 341.598,Z 303.615,A -85,B 0,C 180,E1 -14468.347,E2 -14468.347} C_VEL
LIN {X 0,Y 340.243,Z 376.544,A -85,B 0,C 180,E1 -14469.916,E2 -14469.916} C_VEL
LIN {X 0,Y 339.537,Z 390.4,A -85,B 0,C 180,E1 -14470.464,E2 -14470.464} C_VEL
LIN {X 0,Y 338.659,Z 403.362,A -85,B 0,C 180,E1 -14471.237,E2 -14471.237} C_VEL
LIN {X 0,Y 337.551,Z 415.965,A -85,B 0,C 180,E1 -14472.272,E2 -14472.272} C_VEL
LIN {X 0,Y 336.665,Z 425.915,A -85,B 0,C 180,E1 -14473.32,E2 -14473.32} C_VEL
LIN {X 0,Y 335.668,Z 436.367,A -85,B 0,C 180,E1 -14474.682,E2 -14474.682} C_VEL
LIN {X 0,Y 334.583,Z 446.435,A -85,B 0,C 180,E1 -14476.332,E2 -14476.332} C_VEL
LIN {X 0,Y 333.551,Z 455.321,A -85,B 0,C 180,E1 -14478.146,E2 -14478.146} C_VEL
LIN {X 0,Y 332.887,Z 462.417,A -85,B 0,C 180,E1 -14479.97,E2 -14479.97} C_VEL
LIN {X 0,Y 332.349,Z 468.887,A -85,B 0,C 180,E1 -14482.1,E2 -14482.1} C_VEL
LIN {X 0,Y 332.04,Z 473.669,A -85,B 0,C 180,E1 -14484.187,E2 -14484.187} C_VEL
LIN {X 0,Y 331.963,Z 477.144,A -85,B 0,C 180,E1 -14486.359,E2 -14486.359} C_VEL
LIN {X 0,Y 331.892,Z 478.477,A -85,B 0,C 180,E1 -14487.573,E2 -14487.573} C_VEL
LIN {X 0,Y 331.873,Z 479.415,A -85,B 0,C 180,E1 -14488.787,E2 -14488.787} C_VEL
LIN {X 0,Y 331.893,Z 479.96,A -85,B 0,C 180,E1 -14490,E2 -14490} C_VEL
LIN {X 0,Y 331.872,Z 480.072,A -85,B 0,C 180,E1 -14491.214,E2 -14491.214} C_VEL
LIN {X 0,Y 331.973,Z 479.126,A -85,B 0,C 180,E1 -14493.642,E2 -14493.642} C_VEL
LIN {X 0,Y 332.086,Z 476.849,A -85,B 0,C 180,E1 -14495.892,E2 -14495.892} C_VEL
LIN {X 0,Y 332.459,Z 473.576,A -85,B 0,C 180,E1 -14497.898,E2 -14497.898} C_VEL
LIN {X 0,Y 333.052,Z 469.53,A -85,B 0,C 180,E1 -14499.719,E2 -14499.719} C_VEL
LIN {X 0,Y 334.045,Z 463.334,A -85,B 0,C 180,E1 -14501.838,E2 -14501.838} C_VEL
LIN {X 0,Y 335.113,Z 456.609,A -85,B 0,C 180,E1 -14503.647,E2 -14503.647} C_VEL
LIN {X 0,Y 336.604,Z 448.286,A -85,B 0,C 180,E1 -14505.439,E2 -14505.439} C_VEL
LIN {X 0,Y 337.851,Z 439.75,A -85,B 0,C 180,E1 -14506.932,E2 -14506.932} C_VEL
LIN {X 0,Y 339.479,Z 429.25,A -85,B 0,C 180,E1 -14508.404,E2 -14508.404} C_VEL
LIN {X 0,Y 341.001,Z 418.855,A -85,B 0,C 180,E1 -14509.567,E2 -14509.567} C_VEL
LIN {X 0,Y 342.433,Z 407.427,A -85,B 0,C 180,E1 -14510.577,E2 -14510.577} C_VEL
LIN {X 0,Y 343.743,Z 394.341,A -85,B 0,C 180,E1 -14511.436,E2 -14511.436} C_VEL
LIN {X 0,Y 344.803,Z 381.129,A -85,B 0,C 180,E1 -14512.035,E2 -14512.035} C_VEL
LIN {X 0,Y 345.313,Z 366.493,A -85,B 0,C 180,E1 -14512.434,E2 -14512.434} C_VEL
LIN {X 0,Y 346.796,Z 304.175,A -85,B 0,C 180,E1 -14513.763,E2 -14513.763} C_VEL
LIN {X 0,Y 343.443,Z 286.093,A -85,B 0,C 180,E1 -14514.489,E2 -14514.489} C_VEL
LIN {X 0,Y 339.756,Z 270.776,A -85,B 0,C 180,E1 -14515.21,E2 -14515.21} C_VEL
LIN {X 0,Y 338.678,Z 267.858,A -85,B 0,C 180,E1 -14515.432,E2 -14515.432} C_VEL
LIN {X 0,Y 336.981,Z 259.19,A -85,B 0,C 180,E1 -14517.986,E2 -14517.986} C_VEL
LIN {X 0,Y 334.703,Z 249.607,A -85,B 0,C 180,E1 -14521.055,E2 -14521.055} C_VEL
LIN {X 0,Y 333.669,Z 245.48,A -85,B 0,C 180,E1 -14522.525,E2 -14522.525} C_VEL
LIN {X 0,Y 333.69,Z 245.413,A -85,B 0,C 180,E1 -14526.138,E2 -14526.138} C_VEL
LIN {X 0,Y 333.616,Z 245.418,A -85,B 0,C 180,E1 -14529.197,E2 -14529.197} C_VEL
LIN {X 0,Y 333.643,Z 245.411,A -85,B 0,C 180,E1 -14532.497,E2 -14532.497} C_VEL
LIN {X 0,Y 333.61,Z 245.421,A -85,B 0,C 180,E1 -14535.952,E2 -14535.952} C_VEL
LIN {X 0,Y 333.658,Z 245.423,A -85,B 0,C 180,E1 -14539.314,E2 -14539.314} C_VEL
LIN {X 0,Y 333.675,Z 245.421,A -85,B 0,C 180,E1 -14543.166,E2 -14543.166} C_VEL
LIN {X 0,Y 333.685,Z 245.419,A -85,B 0,C 180,E1 -14545.338,E2 -14545.338} C_VEL
LIN {X 0,Y 333.639,Z 245.418,A -85,B 0,C 180,E1 -14548.218,E2 -14548.218} C_VEL
LIN {X 0,Y 333.662,Z 245.418,A -85,B 0,C 180,E1 -14551.019,E2 -14551.019} C_VEL
LIN {X 0,Y 333.674,Z 245.415,A -85,B 0,C 180,E1 -14555.082,E2 -14555.082} C_VEL
LIN {X 0,Y 333.673,Z 245.418,A -85,B 0,C 180,E1 -14559.014,E2 -14559.014} C_VEL
LIN {X 0,Y 333.75,Z 245.411,A -85,B 0,C 180,E1 -14561.582,E2 -14561.582} C_VEL
LIN {X 0,Y 333.816,Z 245.397,A -85,B 0,C 180,E1 -14565.572,E2 -14565.572} C_VEL
LIN {X 0,Y 333.823,Z 245.392,A -85,B 0,C 180,E1 -14569.073,E2 -14569.073} C_VEL
LIN {X 0,Y 333.976,Z 245.378,A -85,B 0,C 180,E1 -14572.741,E2 -14572.741} C_VEL
LIN {X 0,Y 333.794,Z 245.401,A -85,B 0,C 180,E1 -14575.164,E2 -14575.164} C_VEL
LIN {X 0,Y 334.074,Z 245.367,A -85,B 0,C 180,E1 -14577.583,E2 -14577.583} C_VEL
LIN {X 0,Y 334.207,Z 245.352,A -85,B 0,C 180,E1 -14579.995,E2 -14579.995} C_VEL
LIN {X 0,Y 334.094,Z 245.36,A -85,B 0,C 180,E1 -14582.406,E2 -14582.406} C_VEL
LIN {X 0,Y 333.969,Z 245.378,A -85,B 0,C 180,E1 -14586.486,E2 -14586.486} C_VEL
LIN {X 0,Y 333.844,Z 245.399,A -85,B 0,C 180,E1 -14589.69,E2 -14589.69} C_VEL
LIN {X 0,Y 333.79,Z 245.406,A -85,B 0,C 180,E1 -14593.385,E2 -14593.385} C_VEL
LIN {X 0,Y 333.71,Z 245.416,A -85,B 0,C 180,E1 -14597.142,E2 -14597.142} C_VEL
LIN {X 0,Y 333.71,Z 245.414,A -85,B 0,C 180,E1 -14599.685,E2 -14599.685} C_VEL
LIN {X 0,Y 333.679,Z 245.414,A -85,B 0,C 180,E1 -14602.272,E2 -14602.272} C_VEL
LIN {X 0,Y 333.719,Z 245.394,A -85,B 0,C 180,E1 -14606.24,E2 -14606.24} C_VEL
LIN {X 0,Y 333.672,Z 245.424,A -85,B 0,C 180,E1 -14608.968,E2 -14608.968} C_VEL
LIN {X 0,Y 333.623,Z 245.426,A -85,B 0,C 180,E1 -14612.581,E2 -14612.581} C_VEL
LIN {X 0,Y 333.655,Z 245.42,A -85,B 0,C 180,E1 -14616.133,E2 -14616.133} C_VEL
LIN {X 0,Y 333.662,Z 245.419,A -85,B 0,C 180,E1 -14619.181,E2 -14619.181} C_VEL
LIN {X 0,Y 333.703,Z 245.569,A -85,B 0,C 180,E1 -14621.854,E2 -14621.854} C_VEL
LIN {X 0,Y 335.874,Z 254.41,A -85,B 0,C 180,E1 -14624.82,E2 -14624.82} C_VEL
LIN {X 0,Y 337.084,Z 259.934,A -85,B 0,C 180,E1 -14626.469,E2 -14626.469} C_VEL
LIN {X 0,Y 343.025,Z 273.569,A -85,B 0,C 180,E1 -14627.406,E2 -14627.406} C_VEL
LIN {X 0,Y 346.488,Z 288.922,A -85,B 0,C 180,E1 -14628.088,E2 -14628.088} C_VEL
LIN {X 0,Y 347.129,Z 292.773,A -85,B 0,C 180,E1 -14628.235,E2 -14628.235} C_VEL
LIN {X 0,Y 345.134,Z 368.002,A -85,B 0,C 180,E1 -14629.863,E2 -14629.863} C_VEL
LIN {X 0,Y 344.345,Z 380.982,A -85,B 0,C 180,E1 -14630.371,E2 -14630.371} C_VEL
LIN {X 0,Y 343.245,Z 393.931,A -85,B 0,C 180,E1 -14631.127,E2 -14631.127} C_VEL
LIN {X 0,Y 341.899,Z 406.152,A -85,B 0,C 180,E1 -14632.113,E2 -14632.113} C_VEL
LIN {X 0,Y 340.473,Z 416.922,A -85,B 0,C 180,E1 -14633.229,E2 -14633.229} C_VEL
LIN {X 0,Y 338.837,Z 427.981,A -85,B 0,C 180,E1 -14634.678,E2 -14634.678} C_VEL
LIN {X 0,Y 337.318,Z 437.342,A -85,B 0,C 180,E1 -14636.224,E2 -14636.224} C_VEL
LIN {X 0,Y 335.754,Z 446.425,A -85,B 0,C 180,E1 -14638.093,E2 -14638.093} C_VEL
LIN {X 0,Y 334.434,Z 453.898,A -85,B 0,C 180,E1 -14640.059,E2 -14640.059} C_VEL
LIN {X 0,Y 333.326,Z 460.477,A -85,B 0,C 180,E1 -14642.302,E2 -14642.302} C_VEL
LIN {X 0,Y 332.671,Z 464.9,A -85,B 0,C 180,E1 -14644.336,E2 -14644.336} C_VEL
LIN {X 0,Y 332.179,Z 467.953,A -85,B 0,C 180,E1 -14646.297,E2 -14646.297} C_VEL
LIN {X 0,Y 331.863,Z 470.198,A -85,B 0,C 180,E1 -14648.696,E2 -14648.696} C_VEL
LIN {X 0,Y 331.72,Z 470.831,A -85,B 0,C 180,E1 -14650.185,E2 -14650.185} C_VEL
LIN {X 0,Y 331.701,Z 470.631,A -85,B 0,C 180,E1 -14652.423,E2 -14652.423} C_VEL
LIN {X 0,Y 331.714,Z 469.703,A -85,B 0,C 180,E1 -14654.012,E2 -14654.012} C_VEL
LIN {X 0,Y 331.776,Z 468.433,A -85,B 0,C 180,E1 -14655.274,E2 -14655.274} C_VEL
LIN {X 0,Y 332.007,Z 466.33,A -85,B 0,C 180,E1 -14656.805,E2 -14656.805} C_VEL
LIN {X 0,Y 332.319,Z 461.95,A -85,B 0,C 180,E1 -14659.027,E2 -14659.027} C_VEL
LIN {X 0,Y 332.722,Z 457.033,A -85,B 0,C 180,E1 -14660.884,E2 -14660.884} C_VEL
LIN {X 0,Y 333.35,Z 450.814,A -85,B 0,C 180,E1 -14662.732,E2 -14662.732} C_VEL
LIN {X 0,Y 334.166,Z 443.08,A -85,B 0,C 180,E1 -14664.569,E2 -14664.569} C_VEL
LIN {X 0,Y 334.914,Z 435.173,A -85,B 0,C 180,E1 -14666.089,E2 -14666.089} C_VEL
LIN {X 0,Y 335.967,Z 425.472,A -85,B 0,C 180,E1 -14667.602,E2 -14667.602} C_VEL
LIN {X 0,Y 337.157,Z 414.353,A -85,B 0,C 180,E1 -14668.991,E2 -14668.991} C_VEL
LIN {X 0,Y 338.233,Z 402.499,A -85,B 0,C 180,E1 -14670.148,E2 -14670.148} C_VEL
LIN {X 0,Y 339.048,Z 390.637,A -85,B 0,C 180,E1 -14671.039,E2 -14671.039} C_VEL
LIN {X 0,Y 339.81,Z 377.804,A -85,B 0,C 180,E1 -14671.74,E2 -14671.74} C_VEL
LIN {X 0,Y 340.281,Z 365.407,A -85,B 0,C 180,E1 -14672.182,E2 -14672.182} C_VEL
LIN {X 0,Y 341.658,Z 289.416,A -85,B 0,C 180,E1 -14673.796,E2 -14673.796} C_VEL
LIN {X 0,Y 336.708,Z 260.939,A -85,B 0,C 180,E1 -14674.715,E2 -14674.715} C_VEL
LIN {X 0,Y 336.34,Z 259.387,A -85,B 0,C 180,E1 -14674.869,E2 -14674.869} C_VEL
LIN {X 0,Y 334.657,Z 249.053,A -85,B 0,C 180,E1 -14677.845,E2 -14677.845} C_VEL
LIN {X 0,Y 333.922,Z 245.467,A -85,B 0,C 180,E1 -14678.997,E2 -14678.997} C_VEL
LIN {X 0,Y 333.796,Z 245.406,A -85,B 0,C 180,E1 -14683.391,E2 -14683.391} C_VEL
LIN {X 0,Y 333.719,Z 245.411,A -85,B 0,C 180,E1 -14687.147,E2 -14687.147} C_VEL
LIN {X 0,Y 333.716,Z 245.396,A -85,B 0,C 180,E1 -14689.691,E2 -14689.691} C_VEL
LIN {X 0,Y 333.683,Z 245.415,A -85,B 0,C 180,E1 -14693.449,E2 -14693.449} C_VEL
LIN {X 0,Y 333.048,Z 245.494,A -85,B 0,C 180,E1 -14694.457,E2 -14694.457} C_VEL
LIN {X 0,Y 330.194,Z 245.839,A -85,B 0,C 180,E1 -14696.097,E2 -14696.097} C_VEL
LIN {X 0,Y 327.753,Z 246.134,A -85,B 0,C 180,E1 -14697.426,E2 -14697.426} C_VEL
LIN {X 0,Y 326.701,Z 246.267,A -85,B 0,C 180,E1 -14698.454,E2 -14698.454} C_VEL
LIN {X 0,Y 326.615,Z 246.278,A -85,B 0,C 180,E1 -14698.803,E2 -14698.803} C_VEL
LIN {X 0,Y 326.628,Z 246.299,A -85,B 0,C 180,E1 -14702.541,E2 -14702.541} C_VEL
LIN {X 0,Y 326.632,Z 246.287,A -85,B 0,C 180,E1 -14705.516,E2 -14705.516} C_VEL
LIN {X 0,Y 326.644,Z 246.297,A -85,B 0,C 180,E1 -14709.246,E2 -14709.246} C_VEL
LIN {X 0,Y 326.63,Z 246.279,A -85,B 0,C 180,E1 -14712.993,E2 -14712.993} C_VEL
LIN {X 0,Y 326.631,Z 246.297,A -85,B 0,C 180,E1 -14716.496,E2 -14716.496} C_VEL
LIN {X 0,Y 326.606,Z 246.286,A -85,B 0,C 180,E1 -14719.803,E2 -14719.803} C_VEL
LIN {X 0,Y 326.606,Z 246.287,A -85,B 0,C 180,E1 -14722.959,E2 -14722.959} C_VEL
LIN {X 0,Y 326.598,Z 246.3,A -85,B 0,C 180,E1 -14727.058,E2 -14727.058} C_VEL
LIN {X 0,Y 326.639,Z 246.277,A -85,B 0,C 180,E1 -14730.347,E2 -14730.347} C_VEL
LIN {X 0,Y 326.672,Z 246.274,A -85,B 0,C 180,E1 -14734.522,E2 -14734.522} C_VEL
LIN {X 0,Y 326.645,Z 246.297,A -85,B 0,C 180,E1 -14738.552,E2 -14738.552} C_VEL
LIN {X 0,Y 326.73,Z 246.274,A -85,B 0,C 180,E1 -14741.183,E2 -14741.183} C_VEL
LIN {X 0,Y 326.751,Z 246.248,A -85,B 0,C 180,E1 -14745.439,E2 -14745.439} C_VEL
LIN {X 0,Y 326.764,Z 246.272,A -85,B 0,C 180,E1 -14748.845,E2 -14748.845} C_VEL
LIN {X 0,Y 326.972,Z 246.252,A -85,B 0,C 180,E1 -14752.596,E2 -14752.596} C_VEL
LIN {X 0,Y 326.772,Z 246.265,A -85,B 0,C 180,E1 -14755.071,E2 -14755.071} C_VEL
LIN {X 0,Y 327.041,Z 246.21,A -85,B 0,C 180,E1 -14757.542,E2 -14757.542} C_VEL
LIN {X 0,Y 327.176,Z 246.209,A -85,B 0,C 180,E1 -14760.006,E2 -14760.006} C_VEL
LIN {X 0,Y 327.043,Z 246.243,A -85,B 0,C 180,E1 -14762.469,E2 -14762.469} C_VEL
LIN {X 0,Y 326.952,Z 246.252,A -85,B 0,C 180,E1 -14766.175,E2 -14766.175} C_VEL
LIN {X 0,Y 326.785,Z 246.248,A -85,B 0,C 180,E1 -14769.912,E2 -14769.912} C_VEL
LIN {X 0,Y 326.762,Z 246.273,A -85,B 0,C 180,E1 -14773.69,E2 -14773.69} C_VEL
LIN {X 0,Y 326.704,Z 246.284,A -85,B 0,C 180,E1 -14777.533,E2 -14777.533} C_VEL
LIN {X 0,Y 326.663,Z 246.273,A -85,B 0,C 180,E1 -14780.14,E2 -14780.14} C_VEL
LIN {X 0,Y 326.656,Z 246.29,A -85,B 0,C 180,E1 -14784.133,E2 -14784.133} C_VEL
LIN {X 0,Y 326.683,Z 246.291,A -85,B 0,C 180,E1 -14786.863,E2 -14786.863} C_VEL
LIN {X 0,Y 326.621,Z 246.283,A -85,B 0,C 180,E1 -14790.607,E2 -14790.607} C_VEL
LIN {X 0,Y 326.615,Z 246.301,A -85,B 0,C 180,E1 -14794.023,E2 -14794.023} C_VEL
LIN {X 0,Y 326.632,Z 246.287,A -85,B 0,C 180,E1 -14797.241,E2 -14797.241} C_VEL
LIN {X 0,Y 326.586,Z 246.304,A -85,B 0,C 180,E1 -14801.134,E2 -14801.134} C_VEL
LIN {X 0,Y 326.537,Z 246.274,A -85,B 0,C 180,E1 -14804.745,E2 -14804.745} C_VEL
LIN {X 0,Y 326.574,Z 246.302,A -85,B 0,C 180,E1 -14808.155,E2 -14808.155} C_VEL
LIN {X 0,Y 326.579,Z 246.296,A -85,B 0,C 180,E1 -14811.386,E2 -14811.386} C_VEL
LIN {X 0,Y 326.631,Z 246.297,A -85,B 0,C 180,E1 -14814.854,E2 -14814.854} C_VEL
LIN {X 0,Y 326.621,Z 246.301,A -85,B 0,C 180,E1 -14817.458,E2 -14817.458} C_VEL
LIN {X 0,Y 326.727,Z 246.483,A -85,B 0,C 180,E1 -14820.703,E2 -14820.703} C_VEL
LIN {X 0,Y 328.487,Z 255.234,A -85,B 0,C 180,E1 -14823.302,E2 -14823.302} C_VEL
LIN {X 0,Y 329.953,Z 264.028,A -85,B 0,C 180,E1 -14825.794,E2 -14825.794} C_VEL
LIN {X 0,Y 329.601,Z 268.235,A -85,B 0,C 180,E1 -14826.837,E2 -14826.837} C_VEL
LIN {X 0,Y 331.126,Z 278.565,A -85,B 0,C 180,E1 -14827.208,E2 -14827.208} C_VEL
LIN {X 0,Y 334.84,Z 303.498,A -85,B 0,C 180,E1 -14827.979,E2 -14827.979} C_VEL
LIN {X 0,Y 333.445,Z 376.158,A -85,B 0,C 180,E1 -14829.569,E2 -14829.569} C_VEL
LIN {X 0,Y 332.821,Z 389.364,A -85,B 0,C 180,E1 -14830.093,E2 -14830.093} C_VEL
LIN {X 0,Y 331.909,Z 402.084,A -85,B 0,C 180,E1 -14830.841,E2 -14830.841} C_VEL
LIN {X 0,Y 330.92,Z 413.385,A -85,B 0,C 180,E1 -14831.745,E2 -14831.745} C_VEL
LIN {X 0,Y 329.868,Z 423.774,A -85,B 0,C 180,E1 -14832.806,E2 -14832.806} C_VEL
LIN {X 0,Y 328.836,Z 435.175,A -85,B 0,C 180,E1 -14834.282,E2 -14834.282} C_VEL
LIN {X 0,Y 327.761,Z 444.194,A -85,B 0,C 180,E1 -14835.725,E2 -14835.725} C_VEL
LIN {X 0,Y 326.901,Z 452.098,A -85,B 0,C 180,E1 -14837.27,E2 -14837.27} C_VEL
LIN {X 0,Y 326.085,Z 459.794,A -85,B 0,C 180,E1 -14839.13,E2 -14839.13} C_VEL
LIN {X 0,Y 325.422,Z 466.883,A -85,B 0,C 180,E1 -14841.305,E2 -14841.305} C_VEL
LIN {X 0,Y 325.07,Z 471.573,A -85,B 0,C 180,E1 -14843.171,E2 -14843.171} C_VEL
LIN {X 0,Y 324.894,Z 475.134,A -85,B 0,C 180,E1 -14845.037,E2 -14845.037} C_VEL
LIN {X 0,Y 324.871,Z 476.945,A -85,B 0,C 180,E1 -14846.279,E2 -14846.279} C_VEL
LIN {X 0,Y 324.814,Z 478.301,A -85,B 0,C 180,E1 -14847.52,E2 -14847.52} C_VEL
LIN {X 0,Y 324.785,Z 479.261,A -85,B 0,C 180,E1 -14848.761,E2 -14848.761} C_VEL
LIN {X 0,Y 324.802,Z 479.831,A -85,B 0,C 180,E1 -14850,E2 -14850} C_VEL
LIN {X 0,Y 324.784,Z 479.984,A -85,B 0,C 180,E1 -14851.24,E2 -14851.24} C_VEL
LIN {X 0,Y 324.884,Z 479.081,A -85,B 0,C 180,E1 -14853.721,E2 -14853.721} C_VEL
LIN {X 0,Y 325.009,Z 477.03,A -85,B 0,C 180,E1 -14855.871,E2 -14855.871} C_VEL
LIN {X 0,Y 325.425,Z 473.645,A -85,B 0,C 180,E1 -14858.07,E2 -14858.07} C_VEL
LIN {X 0,Y 326.047,Z 469.65,A -85,B 0,C 180,E1 -14859.93,E2 -14859.93} C_VEL
LIN {X 0,Y 327.088,Z 463.529,A -85,B 0,C 180,E1 -14862.093,E2 -14862.093} C_VEL
LIN {X 0,Y 328.232,Z 456.878,A -85,B 0,C 180,E1 -14863.939,E2 -14863.939} C_VEL
LIN {X 0,Y 329.775,Z 448.643,A -85,B 0,C 180,E1 -14865.767,E2 -14865.767} C_VEL
LIN {X 0,Y 331.09,Z 440.226,A -85,B 0,C 180,E1 -14867.288,E2 -14867.288} C_VEL
LIN {X 0,Y 332.793,Z 429.846,A -85,B 0,C 180,E1 -14868.787,E2 -14868.787} C_VEL
LIN {X 0,Y 334.578,Z 418.186,A -85,B 0,C 180,E1 -14870.119,E2 -14870.119} C_VEL
LIN {X 0,Y 336.098,Z 406.534,A -85,B 0,C 180,E1 -14871.144,E2 -14871.144} C_VEL
LIN {X 0,Y 337.459,Z 393.203,A -85,B 0,C 180,E1 -14872.017,E2 -14872.017} C_VEL
LIN {X 0,Y 338.471,Z 380.421,A -85,B 0,C 180,E1 -14872.59,E2 -14872.59} C_VEL
LIN {X 0,Y 339.027,Z 365.331,A -85,B 0,C 180,E1 -14872.994,E2 -14872.994} C_VEL
LIN {X 0,Y 340.474,Z 304.689,A -85,B 0,C 180,E1 -14874.316,E2 -14874.316} C_VEL
LIN {X 0,Y 336.919,Z 286.041,A -85,B 0,C 180,E1 -14875.108,E2 -14875.108} C_VEL
LIN {X 0,Y 333.915,Z 273.64,A -85,B 0,C 180,E1 -14875.712,E2 -14875.712} C_VEL
LIN {X 0,Y 331.508,Z 267.733,A -85,B 0,C 180,E1 -14876.152,E2 -14876.152} C_VEL
LIN {X 0,Y 330.009,Z 260.1,A -85,B 0,C 180,E1 -14878.463,E2 -14878.463} C_VEL
LIN {X 0,Y 327.331,Z 249.167,A -85,B 0,C 180,E1 -14882.1,E2 -14882.1} C_VEL
LIN {X 0,Y 326.621,Z 246.359,A -85,B 0,C 180,E1 -14883.16,E2 -14883.16} C_VEL
LIN {X 0,Y 326.641,Z 246.299,A -85,B 0,C 180,E1 -14887.046,E2 -14887.046} C_VEL
LIN {X 0,Y 326.559,Z 246.306,A -85,B 0,C 180,E1 -14891.122,E2 -14891.122} C_VEL
LIN {X 0,Y 326.575,Z 246.296,A -85,B 0,C 180,E1 -14893.524,E2 -14893.524} C_VEL
LIN {X 0,Y 326.59,Z 246.283,A -85,B 0,C 180,E1 -14897.026,E2 -14897.026} C_VEL
LIN {X 0,Y 326.613,Z 246.298,A -85,B 0,C 180,E1 -14900.773,E2 -14900.773} C_VEL
LIN {X 0,Y 326.623,Z 246.295,A -85,B 0,C 180,E1 -14904.477,E2 -14904.477} C_VEL
LIN {X 0,Y 326.62,Z 246.294,A -85,B 0,C 180,E1 -14907.452,E2 -14907.452} C_VEL
LIN {X 0,Y 326.626,Z 246.299,A -85,B 0,C 180,E1 -14910.333,E2 -14910.333} C_VEL
LIN {X 0,Y 326.612,Z 246.3,A -85,B 0,C 180,E1 -14914.505,E2 -14914.505} C_VEL
LIN {X 0,Y 326.624,Z 246.298,A -85,B 0,C 180,E1 -14918.539,E2 -14918.539} C_VEL
LIN {X 0,Y 326.673,Z 246.292,A -85,B 0,C 180,E1 -14922.466,E2 -14922.466} C_VEL
LIN {X 0,Y 326.767,Z 246.28,A -85,B 0,C 180,E1 -14926.31,E2 -14926.31} C_VEL
LIN {X 0,Y 326.789,Z 246.273,A -85,B 0,C 180,E1 -14930.088,E2 -14930.088} C_VEL
LIN {X 0,Y 326.958,Z 246.248,A -85,B 0,C 180,E1 -14933.825,E2 -14933.825} C_VEL
LIN {X 0,Y 327.018,Z 246.246,A -85,B 0,C 180,E1 -14937.531,E2 -14937.531} C_VEL
LIN {X 0,Y 327.159,Z 246.23,A -85,B 0,C 180,E1 -14939.994,E2 -14939.994} C_VEL
LIN {X 0,Y 327.035,Z 246.238,A -85,B 0,C 180,E1 -14942.458,E2 -14942.458} C_VEL
LIN {X 0,Y 326.93,Z 246.254,A -85,B 0,C 180,E1 -14946.474,E2 -14946.474} C_VEL
LIN {X 0,Y 326.799,Z 246.278,A -85,B 0,C 180,E1 -14949.901,E2 -14949.901} C_VEL
LIN {X 0,Y 326.752,Z 246.282,A -85,B 0,C 180,E1 -14953.679,E2 -14953.679} C_VEL
LIN {X 0,Y 326.654,Z 246.294,A -85,B 0,C 180,E1 -14957.524,E2 -14957.524} C_VEL
LIN {X 0,Y 326.643,Z 246.296,A -85,B 0,C 180,E1 -14960.129,E2 -14960.129} C_VEL
LIN {X 0,Y 326.638,Z 246.297,A -85,B 0,C 180,E1 -14964.123,E2 -14964.123} C_VEL
LIN {X 0,Y 326.666,Z 246.275,A -85,B 0,C 180,E1 -14966.852,E2 -14966.852} C_VEL
LIN {X 0,Y 326.615,Z 246.287,A -85,B 0,C 180,E1 -14970.604,E2 -14970.604} C_VEL
LIN {X 0,Y 326.585,Z 246.3,A -85,B 0,C 180,E1 -14974.013,E2 -14974.013} C_VEL
LIN {X 0,Y 326.609,Z 246.299,A -85,B 0,C 180,E1 -14977.234,E2 -14977.234} C_VEL
LIN {X 0,Y 326.627,Z 246.35,A -85,B 0,C 180,E1 -14981.141,E2 -14981.141} C_VEL
LIN {X 0,Y 328.14,Z 252.249,A -85,B 0,C 180,E1 -14983.264,E2 -14983.264} C_VEL
LIN {X 0,Y 329.84,Z 259.813,A -85,B 0,C 180,E1 -14985.693,E2 -14985.693} C_VEL
LIN {X 0,Y 331.753,Z 264.115,A -85,B 0,C 180,E1 -14986.066,E2 -14986.066} C_VEL
LIN {X 0,Y 337.294,Z 276.704,A -85,B 0,C 180,E1 -14986.935,E2 -14986.935} C_VEL
LIN {X 0,Y 340.617,Z 292.103,A -85,B 0,C 180,E1 -14987.629,E2 -14987.629} C_VEL
LIN {X 0,Y 340.876,Z 294.788,A -85,B 0,C 180,E1 -14987.718,E2 -14987.718} C_VEL
LIN {X 0,Y 338.844,Z 367.295,A -85,B 0,C 180,E1 -14989.303,E2 -14989.303} C_VEL
LIN {X 0,Y 338.001,Z 380.514,A -85,B 0,C 180,E1 -14989.817,E2 -14989.817} C_VEL
LIN {X 0,Y 336.946,Z 392.883,A -85,B 0,C 180,E1 -14990.537,E2 -14990.537} C_VEL
LIN {X 0,Y 335.623,Z 404.672,A -85,B 0,C 180,E1 -14991.466,E2 -14991.466} C_VEL
LIN {X 0,Y 334.199,Z 415.348,A -85,B 0,C 180,E1 -14992.558,E2 -14992.558} C_VEL
LIN {X 0,Y 332.588,Z 425.907,A -85,B 0,C 180,E1 -14993.911,E2 -14993.911} C_VEL
LIN {X 0,Y 331.044,Z 434.931,A -85,B 0,C 180,E1 -14995.341,E2 -14995.341} C_VEL
LIN {X 0,Y 329.513,Z 443.656,A -85,B 0,C 180,E1 -14997.052,E2 -14997.052} C_VEL
LIN {X 0,Y 327.961,Z 451.728,A -85,B 0,C 180,E1 -14999.049,E2 -14999.049} C_VEL
LIN {X 0,Y 326.797,Z 458.114,A -85,B 0,C 180,E1 -15001.061,E2 -15001.061} C_VEL
LIN {X 0,Y 325.934,Z 463.039,A -85,B 0,C 180,E1 -15003.075,E2 -15003.075} C_VEL
LIN {X 0,Y 325.385,Z 466.687,A -85,B 0,C 180,E1 -15005.097,E2 -15005.097} C_VEL
LIN {X 0,Y 324.943,Z 469.167,A -85,B 0,C 180,E1 -15007.088,E2 -15007.088} C_VEL
LIN {X 0,Y 324.794,Z 470.263,A -85,B 0,C 180,E1 -15008.483,E2 -15008.483} C_VEL
LIN {X 0,Y 324.653,Z 470.847,A -85,B 0,C 180,E1 -15009.735,E2 -15009.735} C_VEL
LIN {X 0,Y 324.598,Z 471.017,A -85,B 0,C 180,E1 -15011.048,E2 -15011.048} C_VEL
LIN {X 0,Y 324.596,Z 470.726,A -85,B 0,C 180,E1 -15012.354,E2 -15012.354} C_VEL
LIN {X 0,Y 324.61,Z 470.025,A -85,B 0,C 180,E1 -15013.652,E2 -15013.652} C_VEL
LIN {X 0,Y 324.648,Z 468.901,A -85,B 0,C 180,E1 -15014.943,E2 -15014.943} C_VEL
LIN {X 0,Y 324.892,Z 466.572,A -85,B 0,C 180,E1 -15016.727,E2 -15016.727} C_VEL
LIN {X 0,Y 325.199,Z 462.761,A -85,B 0,C 180,E1 -15018.784,E2 -15018.784} C_VEL
LIN {X 0,Y 325.573,Z 458.036,A -85,B 0,C 180,E1 -15020.682,E2 -15020.682} C_VEL
LIN {X 0,Y 326.215,Z 452.02,A -85,B 0,C 180,E1 -15022.573,E2 -15022.573} C_VEL
LIN {X 0,Y 326.975,Z 444.536,A -85,B 0,C 180,E1 -15024.449,E2 -15024.449} C_VEL
LIN {X 0,Y 327.779,Z 436.909,A -85,B 0,C 180,E1 -15026.004,E2 -15026.004} C_VEL
LIN {X 0,Y 328.791,Z 427.66,A -85,B 0,C 180,E1 -15027.549,E2 -15027.549} C_VEL
LIN {X 0,Y 329.947,Z 417.479,A -85,B 0,C 180,E1 -15028.913,E2 -15028.913} C_VEL
LIN {X 0,Y 331.089,Z 405.842,A -85,B 0,C 180,E1 -15030.152,E2 -15030.152} C_VEL
LIN {X 0,Y 332,Z 393.962,A -85,B 0,C 180,E1 -15031.137,E2 -15031.137} C_VEL
LIN {X 0,Y 332.782,Z 381.553,A -85,B 0,C 180,E1 -15031.891,E2 -15031.891} C_VEL
LIN {X 0,Y 333.412,Z 367.753,A -85,B 0,C 180,E1 -15032.453,E2 -15032.453} C_VEL
LIN {X 0,Y 334.903,Z 290.368,A -85,B 0,C 180,E1 -15034.145,E2 -15034.145} C_VEL
LIN {X 0,Y 330.278,Z 263.333,A -85,B 0,C 180,E1 -15035.025,E2 -15035.025} C_VEL
LIN {X 0,Y 329.215,Z 259.668,A -85,B 0,C 180,E1 -15035.243,E2 -15035.243} C_VEL
LIN {X 0,Y 327.662,Z 250.245,A -85,B 0,C 180,E1 -15038.014,E2 -15038.014} C_VEL
LIN {X 0,Y 326.856,Z 246.35,A -85,B 0,C 180,E1 -15039.279,E2 -15039.279} C_VEL
LIN {X 0,Y 326.729,Z 246.284,A -85,B 0,C 180,E1 -15042.421,E2 -15042.421} C_VEL
LIN {X 0,Y 326.698,Z 246.29,A -85,B 0,C 180,E1 -15046.239,E2 -15046.239} C_VEL
LIN {X 0,Y 326.72,Z 246.266,A -85,B 0,C 180,E1 -15048.856,E2 -15048.856} C_VEL
LIN {X 0,Y 326.657,Z 246.297,A -85,B 0,C 180,E1 -15052.784,E2 -15052.784} C_VEL
LIN {X 0,Y 326.647,Z 246.26,A -85,B 0,C 180,E1 -15056.86,E2 -15056.86} C_VEL
LIN {X 0,Y 326.615,Z 246.278,A -85,B 0,C 180,E1 -15058.803,E2 -15058.803} C_VEL
LIN {X 0,Y 325.942,Z 246.377,A -85,B 0,C 180,E1 -15059.831,E2 -15059.831} C_VEL
LIN {X 0,Y 323.081,Z 246.745,A -85,B 0,C 180,E1 -15061.505,E2 -15061.505} C_VEL
LIN {X 0,Y 320.663,Z 247.043,A -85,B 0,C 180,E1 -15062.861,E2 -15062.861} C_VEL
LIN {X 0,Y 319.631,Z 247.163,A -85,B 0,C 180,E1 -15063.911,E2 -15063.911} C_VEL
LIN {X 0,Y 319.551,Z 247.17,A -85,B 0,C 180,E1 -15064.266,E2 -15064.266} C_VEL
LIN {X 0,Y 319.6,Z 247.175,A -85,B 0,C 180,E1 -15068.003,E2 -15068.003} C_VEL
LIN {X 0,Y 319.614,Z 247.156,A -85,B 0,C 180,E1 -15071.626,E2 -15071.626} C_VEL
LIN {X 0,Y 319.621,Z 247.167,A -85,B 0,C 180,E1 -15075.291,E2 -15075.291} C_VEL
LIN {X 0,Y 319.554,Z 247.171,A -85,B 0,C 180,E1 -15078.726,E2 -15078.726} C_VEL
LIN {X 0,Y 319.572,Z 247.154,A -85,B 0,C 180,E1 -15082.345,E2 -15082.345} C_VEL
LIN {X 0,Y 319.535,Z 247.178,A -85,B 0,C 180,E1 -15085.129,E2 -15085.129} C_VEL
LIN {X 0,Y 319.551,Z 247.17,A -85,B 0,C 180,E1 -15089.062,E2 -15089.062} C_VEL
LIN {X 0,Y 319.588,Z 247.142,A -85,B 0,C 180,E1 -15092.504,E2 -15092.504} C_VEL
LIN {X 0,Y 319.591,Z 247.167,A -85,B 0,C 180,E1 -15095.31,E2 -15095.31} C_VEL
LIN {X 0,Y 319.614,Z 247.169,A -85,B 0,C 180,E1 -15099.408,E2 -15099.408} C_VEL
LIN {X 0,Y 319.645,Z 247.153,A -85,B 0,C 180,E1 -15102.079,E2 -15102.079} C_VEL
LIN {X 0,Y 319.721,Z 247.129,A -85,B 0,C 180,E1 -15106.014,E2 -15106.014} C_VEL
LIN {X 0,Y 319.751,Z 247.152,A -85,B 0,C 180,E1 -15109.879,E2 -15109.879} C_VEL
LIN {X 0,Y 319.926,Z 247.129,A -85,B 0,C 180,E1 -15112.432,E2 -15112.432} C_VEL
LIN {X 0,Y 319.742,Z 247.142,A -85,B 0,C 180,E1 -15114.962,E2 -15114.962} C_VEL
LIN {X 0,Y 319.985,Z 247.088,A -85,B 0,C 180,E1 -15117.488,E2 -15117.488} C_VEL
LIN {X 0,Y 320.128,Z 247.086,A -85,B 0,C 180,E1 -15120.006,E2 -15120.006} C_VEL
LIN {X 0,Y 319.987,Z 247.122,A -85,B 0,C 180,E1 -15122.523,E2 -15122.523} C_VEL
LIN {X 0,Y 319.909,Z 247.128,A -85,B 0,C 180,E1 -15126.312,E2 -15126.312} C_VEL
LIN {X 0,Y 319.737,Z 247.124,A -85,B 0,C 180,E1 -15130.133,E2 -15130.133} C_VEL
LIN {X 0,Y 319.736,Z 247.15,A -85,B 0,C 180,E1 -15133.997,E2 -15133.997} C_VEL
LIN {X 0,Y 319.663,Z 247.163,A -85,B 0,C 180,E1 -15137.932,E2 -15137.932} C_VEL
LIN {X 0,Y 319.608,Z 247.148,A -85,B 0,C 180,E1 -15140.604,E2 -15140.604} C_VEL
LIN {X 0,Y 319.61,Z 247.173,A -85,B 0,C 180,E1 -15144.701,E2 -15144.701} C_VEL
LIN {X 0,Y 319.614,Z 247.164,A -85,B 0,C 180,E1 -15148.412,E2 -15148.412} C_VEL
LIN {X 0,Y 319.533,Z 247.178,A -85,B 0,C 180,E1 -15151.867,E2 -15151.867} C_VEL
LIN {X 0,Y 319.587,Z 247.171,A -85,B 0,C 180,E1 -15155.546,E2 -15155.546} C_VEL
LIN {X 0,Y 319.57,Z 247.178,A -85,B 0,C 180,E1 -15159.672,E2 -15159.672} C_VEL
LIN {X 0,Y 319.532,Z 247.157,A -85,B 0,C 180,E1 -15163.463,E2 -15163.463} C_VEL
LIN {X 0,Y 319.563,Z 247.16,A -85,B 0,C 180,E1 -15167.019,E2 -15167.019} C_VEL
LIN {X 0,Y 319.543,Z 247.177,A -85,B 0,C 180,E1 -15170.371,E2 -15170.371} C_VEL
LIN {X 0,Y 319.592,Z 247.174,A -85,B 0,C 180,E1 -15174.46,E2 -15174.46} C_VEL
LIN {X 0,Y 319.537,Z 247.179,A -85,B 0,C 180,E1 -15178.139,E2 -15178.139} C_VEL
LIN {X 0,Y 319.659,Z 247.285,A -85,B 0,C 180,E1 -15180.352,E2 -15180.352} C_VEL
LIN {X 0,Y 321.58,Z 256.792,A -85,B 0,C 180,E1 -15183.267,E2 -15183.267} C_VEL
LIN {X 0,Y 322.944,Z 264.754,A -85,B 0,C 180,E1 -15185.577,E2 -15185.577} C_VEL
LIN {X 0,Y 322.719,Z 268.054,A -85,B 0,C 180,E1 -15186.413,E2 -15186.413} C_VEL
LIN {X 0,Y 323.521,Z 273.568,A -85,B 0,C 180,E1 -15186.649,E2 -15186.649} C_VEL
LIN {X 0,Y 328.068,Z 304.703,A -85,B 0,C 180,E1 -15187.632,E2 -15187.632} C_VEL
LIN {X 0,Y 326.656,Z 375.544,A -85,B 0,C 180,E1 -15189.207,E2 -15189.207} C_VEL
LIN {X 0,Y 325.996,Z 388.922,A -85,B 0,C 180,E1 -15189.74,E2 -15189.74} C_VEL
LIN {X 0,Y 325.062,Z 401.73,A -85,B 0,C 180,E1 -15190.503,E2 -15190.503} C_VEL
LIN {X 0,Y 323.979,Z 413.911,A -85,B 0,C 180,E1 -15191.503,E2 -15191.503} C_VEL
LIN {X 0,Y 322.904,Z 424.192,A -85,B 0,C 180,E1 -15192.587,E2 -15192.587} C_VEL
LIN {X 0,Y 321.838,Z 435.498,A -85,B 0,C 180,E1 -15194.091,E2 -15194.091} C_VEL
LIN {X 0,Y 320.643,Z 445.288,A -85,B 0,C 180,E1 -15195.725,E2 -15195.725} C_VEL
LIN {X 0,Y 319.776,Z 452.976,A -85,B 0,C 180,E1 -15197.304,E2 -15197.304} C_VEL
LIN {X 0,Y 318.95,Z 460.496,A -85,B 0,C 180,E1 -15199.205,E2 -15199.205} C_VEL
LIN {X 0,Y 318.382,Z 466.522,A -85,B 0,C 180,E1 -15201.112,E2 -15201.112} C_VEL
LIN {X 0,Y 318.004,Z 471.27,A -85,B 0,C 180,E1 -15203.019,E2 -15203.019} C_VEL
LIN {X 0,Y 317.809,Z 474.883,A -85,B 0,C 180,E1 -15204.926,E2 -15204.926} C_VEL
LIN {X 0,Y 317.782,Z 476.739,A -85,B 0,C 180,E1 -15206.196,E2 -15206.196} C_VEL
LIN {X 0,Y 317.737,Z 478.123,A -85,B 0,C 180,E1 -15207.465,E2 -15207.465} C_VEL
LIN {X 0,Y 317.7,Z 479.105,A -85,B 0,C 180,E1 -15208.733,E2 -15208.733} C_VEL
LIN {X 0,Y 317.713,Z 479.698,A -85,B 0,C 180,E1 -15210,E2 -15210} C_VEL
LIN {X 0,Y 317.699,Z 479.894,A -85,B 0,C 180,E1 -15211.268,E2 -15211.268} C_VEL
LIN {X 0,Y 317.738,Z 479.66,A -85,B 0,C 180,E1 -15212.536,E2 -15212.536} C_VEL
LIN {X 0,Y 317.797,Z 479.041,A -85,B 0,C 180,E1 -15213.804,E2 -15213.804} C_VEL
LIN {X 0,Y 317.985,Z 476.639,A -85,B 0,C 180,E1 -15216.345,E2 -15216.345} C_VEL
LIN {X 0,Y 318.389,Z 473.714,A -85,B 0,C 180,E1 -15218.25,E2 -15218.25} C_VEL
LIN {X 0,Y 319.039,Z 469.77,A -85,B 0,C 180,E1 -15220.151,E2 -15220.151} C_VEL
LIN {X 0,Y 319.978,Z 464.712,A -85,B 0,C 180,E1 -15222.044,E2 -15222.044} C_VEL
LIN {X 0,Y 321.1,Z 458.372,A -85,B 0,C 180,E1 -15223.932,E2 -15223.932} C_VEL
LIN {X 0,Y 322.685,Z 450.463,A -85,B 0,C 180,E1 -15225.798,E2 -15225.798} C_VEL
LIN {X 0,Y 324.066,Z 442.208,A -85,B 0,C 180,E1 -15227.393,E2 -15227.393} C_VEL
LIN {X 0,Y 325.713,Z 432.672,A -85,B 0,C 180,E1 -15228.885,E2 -15228.885} C_VEL
LIN {X 0,Y 327.564,Z 421.764,A -85,B 0,C 180,E1 -15230.241,E2 -15230.241} C_VEL
LIN {X 0,Y 329.292,Z 409.376,A -85,B 0,C 180,E1 -15231.438,E2 -15231.438} C_VEL
LIN {X 0,Y 330.742,Z 397.215,A -85,B 0,C 180,E1 -15232.323,E2 -15232.323} C_VEL
LIN {X 0,Y 331.858,Z 385.32,A -85,B 0,C 180,E1 -15232.943,E2 -15232.943} C_VEL
LIN {X 0,Y 332.559,Z 372.498,A -85,B 0,C 180,E1 -15233.385,E2 -15233.385} C_VEL
LIN {X 0,Y 334.251,Z 305.839,A -85,B 0,C 180,E1 -15234.877,E2 -15234.877} C_VEL
LIN {X 0,Y 331.207,Z 289.429,A -85,B 0,C 180,E1 -15235.586,E2 -15235.586} C_VEL
LIN {X 0,Y 328.199,Z 276.708,A -85,B 0,C 180,E1 -15236.217,E2 -15236.217} C_VEL
LIN {X 0,Y 324.388,Z 267.666,A -85,B 0,C 180,E1 -15236.898,E2 -15236.898} C_VEL
LIN {X 0,Y 322.536,Z 259.071,A -85,B 0,C 180,E1 -15239.617,E2 -15239.617} C_VEL
LIN {X 0,Y 320.149,Z 249.575,A -85,B 0,C 180,E1 -15242.91,E2 -15242.91} C_VEL
LIN {X 0,Y 319.592,Z 247.202,A -85,B 0,C 180,E1 -15243.87,E2 -15243.87} C_VEL
LIN {X 0,Y 319.556,Z 247.176,A -85,B 0,C 180,E1 -15247.645,E2 -15247.645} C_VEL
LIN {X 0,Y 319.52,Z 247.176,A -85,B 0,C 180,E1 -15251.59,E2 -15251.59} C_VEL
LIN {X 0,Y 319.502,Z 247.189,A -85,B 0,C 180,E1 -15254.741,E2 -15254.741} C_VEL
LIN {X 0,Y 319.538,Z 247.167,A -85,B 0,C 180,E1 -15258.401,E2 -15258.401} C_VEL
LIN {X 0,Y 319.548,Z 247.176,A -85,B 0,C 180,E1 -15261.983,E2 -15261.983} C_VEL
LIN {X 0,Y 319.572,Z 247.175,A -85,B 0,C 180,E1 -15265.12,E2 -15265.12} C_VEL
LIN {X 0,Y 319.535,Z 247.174,A -85,B 0,C 180,E1 -15268.134,E2 -15268.134} C_VEL
LIN {X 0,Y 319.582,Z 247.168,A -85,B 0,C 180,E1 -15271.601,E2 -15271.601} C_VEL
LIN {X 0,Y 319.538,Z 247.174,A -85,B 0,C 180,E1 -15275.294,E2 -15275.294} C_VEL
LIN {X 0,Y 319.575,Z 247.176,A -85,B 0,C 180,E1 -15278.041,E2 -15278.041} C_VEL
LIN {X 0,Y 319.623,Z 247.171,A -85,B 0,C 180,E1 -15282.066,E2 -15282.066} C_VEL
LIN {X 0,Y 319.74,Z 247.156,A -85,B 0,C 180,E1 -15286.003,E2 -15286.003} C_VEL
LIN {X 0,Y 319.741,Z 247.149,A -85,B 0,C 180,E1 -15289.867,E2 -15289.867} C_VEL
LIN {X 0,Y 319.914,Z 247.125,A -85,B 0,C 180,E1 -15293.688,E2 -15293.688} C_VEL
LIN {X 0,Y 319.964,Z 247.125,A -85,B 0,C 180,E1 -15297.477,E2 -15297.477} C_VEL
LIN {X 0,Y 320.112,Z 247.107,A -85,B 0,C 180,E1 -15299.994,E2 -15299.994} C_VEL
LIN {X 0,Y 319.978,Z 247.117,A -85,B 0,C 180,E1 -15302.512,E2 -15302.512} C_VEL
LIN {X 0,Y 319.893,Z 247.131,A -85,B 0,C 180,E1 -15306.455,E2 -15306.455} C_VEL
LIN {X 0,Y 319.746,Z 247.156,A -85,B 0,C 180,E1 -15310.121,E2 -15310.121} C_VEL
LIN {X 0,Y 319.725,Z 247.159,A -85,B 0,C 180,E1 -15313.986,E2 -15313.986} C_VEL
LIN {X 0,Y 319.614,Z 247.171,A -85,B 0,C 180,E1 -15317.923,E2 -15317.923} C_VEL
LIN {X 0,Y 319.597,Z 247.177,A -85,B 0,C 180,E1 -15320.593,E2 -15320.593} C_VEL
LIN {X 0,Y 319.557,Z 247.181,A -85,B 0,C 180,E1 -15323.313,E2 -15323.313} C_VEL
LIN {X 0,Y 319.602,Z 247.152,A -85,B 0,C 180,E1 -15326.083,E2 -15326.083} C_VEL
LIN {X 0,Y 319.563,Z 247.181,A -85,B 0,C 180,E1 -15328.928,E2 -15328.928} C_VEL
LIN {X 0,Y 319.51,Z 247.174,A -85,B 0,C 180,E1 -15331.856,E2 -15331.856} C_VEL
LIN {X 0,Y 319.558,Z 247.17,A -85,B 0,C 180,E1 -15335.537,E2 -15335.537} C_VEL
LIN {X 0,Y 319.578,Z 247.168,A -85,B 0,C 180,E1 -15337.998,E2 -15337.998} C_VEL
LIN {X 0,Y 319.618,Z 247.302,A -85,B 0,C 180,E1 -15340.534,E2 -15340.534} C_VEL
LIN {X 0,Y 321.548,Z 255.007,A -85,B 0,C 180,E1 -15343.309,E2 -15343.309} C_VEL
LIN {X 0,Y 322.717,Z 259.975,A -85,B 0,C 180,E1 -15344.933,E2 -15344.933} C_VEL
LIN {X 0,Y 325.127,Z 265.397,A -85,B 0,C 180,E1 -15345.404,E2 -15345.404} C_VEL
LIN {X 0,Y 331.461,Z 279.392,A -85,B 0,C 180,E1 -15346.423,E2 -15346.423} C_VEL
LIN {X 0,Y 334.625,Z 294.429,A -85,B 0,C 180,E1 -15347.113,E2 -15347.113} C_VEL
LIN {X 0,Y 332.502,Z 368.138,A -85,B 0,C 180,E1 -15348.767,E2 -15348.767} C_VEL
LIN {X 0,Y 331.578,Z 381.855,A -85,B 0,C 180,E1 -15349.327,E2 -15349.327} C_VEL
LIN {X 0,Y 330.484,Z 393.782,A -85,B 0,C 180,E1 -15350.052,E2 -15350.052} C_VEL
LIN {X 0,Y 329.153,Z 404.936,A -85,B 0,C 180,E1 -15350.959,E2 -15350.959} C_VEL
LIN {X 0,Y 327.657,Z 415.66,A -85,B 0,C 180,E1 -15352.08,E2 -15352.08} C_VEL
LIN {X 0,Y 325.978,Z 426.09,A -85,B 0,C 180,E1 -15353.445,E2 -15353.445} C_VEL
LIN {X 0,Y 324.319,Z 435.391,A -85,B 0,C 180,E1 -15354.953,E2 -15354.953} C_VEL
LIN {X 0,Y 322.758,Z 443.807,A -85,B 0,C 180,E1 -15356.645,E2 -15356.645} C_VEL
LIN {X 0,Y 321.215,Z 451.429,A -85,B 0,C 180,E1 -15358.557,E2 -15358.557} C_VEL
LIN {X 0,Y 320.053,Z 457.273,A -85,B 0,C 180,E1 -15360.391,E2 -15360.391} C_VEL
LIN {X 0,Y 319.09,Z 462.417,A -85,B 0,C 180,E1 -15362.449,E2 -15362.449} C_VEL
LIN {X 0,Y 318.367,Z 466.745,A -85,B 0,C 180,E1 -15364.815,E2 -15364.815} C_VEL
LIN {X 0,Y 317.928,Z 468.942,A -85,B 0,C 180,E1 -15366.553,E2 -15366.553} C_VEL
LIN {X 0,Y 317.697,Z 470.343,A -85,B 0,C 180,E1 -15368.275,E2 -15368.275} C_VEL
LIN {X 0,Y 317.5,Z 471.113,A -85,B 0,C 180,E1 -15370.608,E2 -15370.608} C_VEL
LIN {X 0,Y 317.49,Z 470.882,A -85,B 0,C 180,E1 -15372.121,E2 -15372.121} C_VEL
LIN {X 0,Y 317.534,Z 469.298,A -85,B 0,C 180,E1 -15374.597,E2 -15374.597} C_VEL
LIN {X 0,Y 317.791,Z 466.817,A -85,B 0,C 180,E1 -15376.636,E2 -15376.636} C_VEL
LIN {X 0,Y 318.06,Z 463.49,A -85,B 0,C 180,E1 -15378.529,E2 -15378.529} C_VEL
LIN {X 0,Y 318.412,Z 458.966,A -85,B 0,C 180,E1 -15380.471,E2 -15380.471} C_VEL
LIN {X 0,Y 319.111,Z 452.545,A -85,B 0,C 180,E1 -15382.593,E2 -15382.593} C_VEL
LIN {X 0,Y 319.958,Z 444.576,A -85,B 0,C 180,E1 -15384.643,E2 -15384.643} C_VEL
LIN {X 0,Y 320.795,Z 436.933,A -85,B 0,C 180,E1 -15386.231,E2 -15386.231} C_VEL
LIN {X 0,Y 321.859,Z 427.658,A -85,B 0,C 180,E1 -15387.81,E2 -15387.81} C_VEL
LIN {X 0,Y 323.109,Z 416.82,A -85,B 0,C 180,E1 -15389.276,E2 -15389.276} C_VEL
LIN {X 0,Y 324.208,Z 405.788,A -85,B 0,C 180,E1 -15390.465,E2 -15390.465} C_VEL
LIN {X 0,Y 325.169,Z 393.849,A -85,B 0,C 180,E1 -15391.47,E2 -15391.47} C_VEL
LIN {X 0,Y 325.976,Z 381.346,A -85,B 0,C 180,E1 -15392.239,E2 -15392.239} C_VEL
LIN {X 0,Y 326.597,Z 368.503,A -85,B 0,C 180,E1 -15392.775,E2 -15392.775} C_VEL
LIN {X 0,Y 327.385,Z 332.103,A -85,B 0,C 180,E1 -15393.615,E2 -15393.615} C_VEL
LIN {X 0,Y 328.109,Z 290.83,A -85,B 0,C 180,E1 -15394.523,E2 -15394.523} C_VEL
LIN {X 0,Y 323.601,Z 264.786,A -85,B 0,C 180,E1 -15395.398,E2 -15395.398} C_VEL
LIN {X 0,Y 322.062,Z 259.907,A -85,B 0,C 180,E1 -15395.655,E2 -15395.655} C_VEL
LIN {X 0,Y 320.684,Z 251.398,A -85,B 0,C 180,E1 -15398.189,E2 -15398.189} C_VEL
LIN {X 0,Y 319.803,Z 247.232,A -85,B 0,C 180,E1 -15399.566,E2 -15399.566} C_VEL
LIN {X 0,Y 319.71,Z 247.159,A -85,B 0,C 180,E1 -15403.993,E2 -15403.993} C_VEL
LIN {X 0,Y 319.623,Z 247.159,A -85,B 0,C 180,E1 -15407.928,E2 -15407.928} C_VEL
LIN {X 0,Y 319.6,Z 247.16,A -85,B 0,C 180,E1 -15410.599,E2 -15410.599} C_VEL
LIN {X 0,Y 319.602,Z 247.171,A -85,B 0,C 180,E1 -15413.316,E2 -15413.316} C_VEL
LIN {X 0,Y 319.596,Z 247.141,A -85,B 0,C 180,E1 -15416.091,E2 -15416.091} C_VEL
LIN {X 0,Y 319.569,Z 247.158,A -85,B 0,C 180,E1 -15418.935,E2 -15418.935} C_VEL
LIN {X 0,Y 319.548,Z 247.183,A -85,B 0,C 180,E1 -15421.859,E2 -15421.859} C_VEL
LIN {X 0,Y 319.551,Z 247.17,A -85,B 0,C 180,E1 -15424.266,E2 -15424.266} C_VEL
LIN {X 0,Y 318.89,Z 247.251,A -85,B 0,C 180,E1 -15425.319,E2 -15425.319} C_VEL
LIN {X 0,Y 316.037,Z 247.612,A -85,B 0,C 180,E1 -15427.033,E2 -15427.033} C_VEL
LIN {X 0,Y 313.626,Z 247.917,A -85,B 0,C 180,E1 -15428.422,E2 -15428.422} C_VEL
LIN {X 0,Y 312.606,Z 248.045,A -85,B 0,C 180,E1 -15429.498,E2 -15429.498} C_VEL
LIN {X 0,Y 312.532,Z 248.048,A -85,B 0,C 180,E1 -15429.862,E2 -15429.862} C_VEL
LIN {X 0,Y 312.546,Z 248.032,A -85,B 0,C 180,E1 -15432.421,E2 -15432.421} C_VEL
LIN {X 0,Y 312.565,Z 248.052,A -85,B 0,C 180,E1 -15436.014,E2 -15436.014} C_VEL
LIN {X 0,Y 312.502,Z 248.04,A -85,B 0,C 180,E1 -15439.874,E2 -15439.874} C_VEL
LIN {X 0,Y 312.526,Z 248.035,A -85,B 0,C 180,E1 -15442.624,E2 -15442.624} C_VEL
LIN {X 0,Y 312.495,Z 248.061,A -85,B 0,C 180,E1 -15446.317,E2 -15446.317} C_VEL
LIN {X 0,Y 312.524,Z 248.034,A -85,B 0,C 180,E1 -15450.356,E2 -15450.356} C_VEL
LIN {X 0,Y 312.584,Z 248.024,A -85,B 0,C 180,E1 -15454.07,E2 -15454.07} C_VEL
LIN {X 0,Y 312.572,Z 248.047,A -85,B 0,C 180,E1 -15457.535,E2 -15457.535} C_VEL
LIN {X 0,Y 312.625,Z 248.028,A -85,B 0,C 180,E1 -15461.663,E2 -15461.663} C_VEL
LIN {X 0,Y 312.682,Z 248.001,A -85,B 0,C 180,E1 -15465.692,E2 -15465.692} C_VEL
LIN {X 0,Y 312.695,Z 248.033,A -85,B 0,C 180,E1 -15469.648,E2 -15469.648} C_VEL
LIN {X 0,Y 312.865,Z 248.009,A -85,B 0,C 180,E1 -15472.26,E2 -15472.26} C_VEL
LIN {X 0,Y 312.712,Z 248.019,A -85,B 0,C 180,E1 -15474.848,E2 -15474.848} C_VEL
LIN {X 0,Y 312.985,Z 247.964,A -85,B 0,C 180,E1 -15478.719,E2 -15478.719} C_VEL
LIN {X 0,Y 312.986,Z 247.985,A -85,B 0,C 180,E1 -15481.292,E2 -15481.292} C_VEL
LIN {X 0,Y 312.705,Z 248.03,A -85,B 0,C 180,E1 -15485.163,E2 -15485.163} C_VEL
LIN {X 0,Y 312.803,Z 248.004,A -85,B 0,C 180,E1 -15487.753,E2 -15487.753} C_VEL
LIN {X 0,Y 312.666,Z 248.012,A -85,B 0,C 180,E1 -15491.677,E2 -15491.677} C_VEL
LIN {X 0,Y 312.704,Z 248.031,A -85,B 0,C 180,E1 -15494.893,E2 -15494.893} C_VEL
LIN {X 0,Y 312.615,Z 248.028,A -85,B 0,C 180,E1 -15499.23,E2 -15499.23} C_VEL
LIN {X 0,Y 312.532,Z 248.041,A -85,B 0,C 180,E1 -15502.785,E2 -15502.785} C_VEL
LIN {X 0,Y 312.603,Z 248.045,A -85,B 0,C 180,E1 -15505.937,E2 -15505.937} C_VEL
LIN {X 0,Y 312.516,Z 248.036,A -85,B 0,C 180,E1 -15509.658,E2 -15509.658} C_VEL
LIN {X 0,Y 312.529,Z 248.056,A -85,B 0,C 180,E1 -15513.693,E2 -15513.693} C_VEL
LIN {X 0,Y 312.524,Z 248.044,A -85,B 0,C 180,E1 -15517.391,E2 -15517.391} C_VEL
LIN {X 0,Y 312.5,Z 248.058,A -85,B 0,C 180,E1 -15520.713,E2 -15520.713} C_VEL
LIN {X 0,Y 312.462,Z 248.029,A -85,B 0,C 180,E1 -15524.213,E2 -15524.213} C_VEL
LIN {X 0,Y 312.467,Z 248.054,A -85,B 0,C 180,E1 -15527.928,E2 -15527.928} C_VEL
LIN {X 0,Y 312.488,Z 248.048,A -85,B 0,C 180,E1 -15531.927,E2 -15531.927} C_VEL
LIN {X 0,Y 312.543,Z 248.054,A -85,B 0,C 180,E1 -15534.223,E2 -15534.223} C_VEL
LIN {X 0,Y 312.515,Z 248.058,A -85,B 0,C 180,E1 -15537.336,E2 -15537.336} C_VEL
LIN {X 0,Y 312.607,Z 248.219,A -85,B 0,C 180,E1 -15540.079,E2 -15540.079} C_VEL
LIN {X 0,Y 314.693,Z 258.589,A -85,B 0,C 180,E1 -15543.3,E2 -15543.3} C_VEL
LIN {X 0,Y 315.956,Z 266.02,A -85,B 0,C 180,E1 -15545.503,E2 -15545.503} C_VEL
LIN {X 0,Y 315.834,Z 268.177,A -85,B 0,C 180,E1 -15546.007,E2 -15546.007} C_VEL
LIN {X 0,Y 320.223,Z 297.626,A -85,B 0,C 180,E1 -15547.016,E2 -15547.016} C_VEL
LIN {X 0,Y 321.322,Z 305.543,A -85,B 0,C 180,E1 -15547.266,E2 -15547.266} C_VEL
LIN {X 0,Y 319.835,Z 376.093,A -85,B 0,C 180,E1 -15548.869,E2 -15548.869} C_VEL
LIN {X 0,Y 319.163,Z 389.251,A -85,B 0,C 180,E1 -15549.413,E2 -15549.413} C_VEL
LIN {X 0,Y 318.244,Z 401.38,A -85,B 0,C 180,E1 -15550.152,E2 -15550.152} C_VEL
LIN {X 0,Y 317.225,Z 412.835,A -85,B 0,C 180,E1 -15551.095,E2 -15551.095} C_VEL
LIN {X 0,Y 315.938,Z 424.601,A -85,B 0,C 180,E1 -15552.357,E2 -15552.357} C_VEL
LIN {X 0,Y 314.842,Z 435.815,A -85,B 0,C 180,E1 -15553.894,E2 -15553.894} C_VEL
LIN {X 0,Y 313.715,Z 444.687,A -85,B 0,C 180,E1 -15555.403,E2 -15555.403} C_VEL
LIN {X 0,Y 312.625,Z 453.829,A -85,B 0,C 180,E1 -15557.339,E2 -15557.339} C_VEL
LIN {X 0,Y 311.805,Z 461.181,A -85,B 0,C 180,E1 -15559.284,E2 -15559.284} C_VEL
LIN {X 0,Y 311.32,Z 466.145,A -85,B 0,C 180,E1 -15560.908,E2 -15560.908} C_VEL
LIN {X 0,Y 310.935,Z 470.953,A -85,B 0,C 180,E1 -15562.859,E2 -15562.859} C_VEL
LIN {X 0,Y 310.715,Z 474.622,A -85,B 0,C 180,E1 -15564.81,E2 -15564.81} C_VEL
LIN {X 0,Y 310.697,Z 476.515,A -85,B 0,C 180,E1 -15566.109,E2 -15566.109} C_VEL
LIN {X 0,Y 310.662,Z 477.939,A -85,B 0,C 180,E1 -15567.407,E2 -15567.407} C_VEL
LIN {X 0,Y 310.617,Z 478.946,A -85,B 0,C 180,E1 -15568.704,E2 -15568.704} C_VEL
LIN {X 0,Y 310.627,Z 479.563,A -85,B 0,C 180,E1 -15570,E2 -15570} C_VEL
LIN {X 0,Y 310.616,Z 479.793,A -85,B 0,C 180,E1 -15571.297,E2 -15571.297} C_VEL
LIN {X 0,Y 310.663,Z 479.597,A -85,B 0,C 180,E1 -15572.594,E2 -15572.594} C_VEL
LIN {X 0,Y 310.713,Z 479.002,A -85,B 0,C 180,E1 -15573.891,E2 -15573.891} C_VEL
LIN {X 0,Y 310.919,Z 476.656,A -85,B 0,C 180,E1 -15576.49,E2 -15576.49} C_VEL
LIN {X 0,Y 311.338,Z 473.775,A -85,B 0,C 180,E1 -15578.438,E2 -15578.438} C_VEL
LIN {X 0,Y 312.031,Z 469.884,A -85,B 0,C 180,E1 -15580.381,E2 -15580.381} C_VEL
LIN {X 0,Y 313.028,Z 464.885,A -85,B 0,C 180,E1 -15582.316,E2 -15582.316} C_VEL
LIN {X 0,Y 314.233,Z 458.632,A -85,B 0,C 180,E1 -15584.243,E2 -15584.243} C_VEL
LIN {X 0,Y 315.873,Z 450.824,A -85,B 0,C 180,E1 -15586.148,E2 -15586.148} C_VEL
LIN {X 0,Y 317.246,Z 443.07,A -85,B 0,C 180,E1 -15587.704,E2 -15587.704} C_VEL
LIN {X 0,Y 319.035,Z 433.26,A -85,B 0,C 180,E1 -15589.295,E2 -15589.295} C_VEL
LIN {X 0,Y 320.966,Z 422.551,A -85,B 0,C 180,E1 -15590.676,E2 -15590.676} C_VEL
LIN {X 0,Y 322.516,Z 412.156,A -85,B 0,C 180,E1 -15591.744,E2 -15591.744} C_VEL
LIN {X 0,Y 324.151,Z 399.678,A -85,B 0,C 180,E1 -15592.718,E2 -15592.718} C_VEL
LIN {X 0,Y 325.442,Z 386.563,A -85,B 0,C 180,E1 -15593.464,E2 -15593.464} C_VEL
LIN {X 0,Y 326.288,Z 373.26,A -85,B 0,C 180,E1 -15593.947,E2 -15593.947} C_VEL
LIN {X 0,Y 328.077,Z 306.854,A -85,B 0,C 180,E1 -15595.461,E2 -15595.461} C_VEL
LIN {X 0,Y 324.886,Z 290.092,A -85,B 0,C 180,E1 -15596.218,E2 -15596.218} C_VEL
LIN {X 0,Y 322.36,Z 279.316,A -85,B 0,C 180,E1 -15596.77,E2 -15596.77} C_VEL
LIN {X 0,Y 317.18,Z 267.568,A -85,B 0,C 180,E1 -15597.71,E2 -15597.71} C_VEL
LIN {X 0,Y 315.796,Z 261.159,A -85,B 0,C 180,E1 -15599.773,E2 -15599.773} C_VEL
LIN {X 0,Y 313.33,Z 251.365,A -85,B 0,C 180,E1 -15603.256,E2 -15603.256} C_VEL
